//Intern Errors
IF bErrorIntern AND iErrorCode = 1 THEN
	eMessageKNXMaster := E_Message_KNXMaster.eTooMuchKNXMasters;
END_IF
//KNX Errors
IF bErrorKNX AND iErrorCode = 1 THEN
	eMessageKNXMaster := E_Message_KNXMaster.eWrong_KNX_Phys_Addr;
ELSIF bErrorKNX AND iErrorCode = 2 THEN
	eMessageKNXMaster := E_Message_KNXMaster.eWrong_KNX_Group_Addr;
ELSIF bErrorKNX AND iErrorCode = 3 THEN
	eMessageKNXMaster := E_Message_KNXMaster.eWrong_KNX_Group_Len;
ELSIF bErrorKNX AND iErrorCode = 4 THEN
	eMessageKNXMaster := E_Message_KNXMaster.eWrong_KNX_No_Filter;
ELSIF bErrorKNX AND iErrorCode = 10 THEN
	eMessageKNXMaster := E_Message_KNXMaster.eWrong_KNX_Firmware;
ELSIF bErrorKNX AND iErrorCode = 11 THEN
	eMessageKNXMaster := E_Message_KNXMaster.eWrong_KNX_Mode;
ELSIF bErrorKNX AND iErrorCode = 12 THEN
	eMessageKNXMaster := E_Message_KNXMaster.eWrong_Mode;
ELSIF bErrorKNX AND iErrorCode = 14 THEN
	eMessageKNXMaster := E_Message_KNXMaster.eWrong_KNX_Firmware_B1_Necessary;
ELSIF bErrorKNX AND iErrorCode = 15 THEN
	eMessageKNXMaster := E_Message_KNXMaster.eWrong_KNX_Firmware_B3_Necessary;
ELSIF bErrorKNX AND iErrorCode = 20 THEN
	eMessageKNXMaster := E_Message_KNXMaster.eWrong_KNX_Data_Len;
ELSIF bErrorKNX AND iErrorCode = 21 THEN
	eMessageKNXMaster := E_Message_KNXMaster.eError_KNX_Service_Not_Support;
ELSIF bErrorKNX AND iErrorCode = 30 THEN
	eMessageKNXMaster := E_Message_KNXMaster.eKL6301_TP_Toggle_Error;
ELSIF bErrorKNX AND iErrorCode = 31 THEN
	eMessageKNXMaster := E_Message_KNXMaster.eTime_Out;
ELSIF bErrorKNX AND iErrorCode = 32 THEN
	eMessageKNXMaster := E_Message_KNXMaster.eKL6301_No_Response_from_Terminal;
ELSIF bErrorKNX AND iErrorCode = 40 THEN
	eMessageKNXMaster := E_Message_KNXMaster.eError_Send_8Bit_Wrong_Scaling_Mode;
ELSIF bErrorKNX AND iErrorCode = 100 THEN
	eMessageKNXMaster := E_Message_KNXMaster.eError_KNX_Phy_Addr_Not_Support;
ELSIF bErrorKNX AND iErrorCode = 101 THEN
	eMessageKNXMaster := E_Message_KNXMaster.eError_KNX_Write_Data;
ELSIF bErrorKNX AND iErrorCode = 102 THEN
	eMessageKNXMaster := E_Message_KNXMaster.eMonitor_Mode_Len_Is_Not_Ok_Must_0;
ELSIF bErrorKNX AND iErrorCode = 103 THEN
	eMessageKNXMaster := E_Message_KNXMaster.eMonitor_Mode_Addr_Is_Not_Ok_Must_0;
ELSIF bErrorKNX AND iErrorCode = 104 THEN
	eMessageKNXMaster := E_Message_KNXMaster.eWatchdog_Error_No_Send;
ELSIF bErrorKNX AND iErrorCode = 16#0BBB THEN
	eMessageKNXMaster := E_Message_KNXMaster.eError_KNX_No_Ack;
ELSIF bErrorKNX AND iErrorCode = 16#FAFB THEN
	eMessageKNXMaster := E_Message_KNXMaster.eError_KNX_No_Com_To_TP;
ELSIF bErrorKNX AND iErrorCode = 16#0FCC THEN
	eMessageKNXMaster := E_Message_KNXMaster.eError_TP_Temp_Warning;
ELSIF bErrorKNX AND iErrorCode = 16#17CC THEN
	eMessageKNXMaster := E_Message_KNXMaster.eError_TP_Protocol_Error;
ELSIF bErrorKNX AND iErrorCode = 16#27CC THEN
	eMessageKNXMaster := E_Message_KNXMaster.eError_TP_Transmitter_Error;
ELSIF bErrorKNX AND iErrorCode = 16#47CC THEN
	eMessageKNXMaster := E_Message_KNXMaster.eError_TP_Receive_Error;
ELSIF bErrorKNX AND iErrorCode = 16#87CC THEN
	eMessageKNXMaster := E_Message_KNXMaster.eError_TP_Slave_Collision;
END_IF 

IF bWarning THEN 
	byErrorWarning := 1;
END_IF	
	IF bErrorKNX OR bErrorIntern THEN
		byErrorWarning := 2;
	END_IF

//All ok
IF NOT bErrorKNX AND NOT bErrorIntern AND NOT bWarning THEN
	eMessageKNXMaster := E_Message_KNXMaster.eAllOk;
		byErrorWarning := 0;
END_IF

END_FUNCTION_BLOCK

// ---- Bussystems/FBs Internal/MBus Master/FB_MBusMaster_Messages.TcPOU
{attribute 'conditionalshow'}
FUNCTION_BLOCK FB_MBusMaster_Messages
VAR_INPUT
	{attribute 'hide'}
	bErrorMBus							: BOOL;						//Error from the Mbus Function
	{attribute 'hide'}
	bErrorIntern						: BOOL;						//Internal Error
	{attribute 'hide'}
	bWarning							: BOOL;						//Warning from the RTU Function
	{attribute 'hide'}
	iWarningCode						: INT;						//Warning Code
	{attribute 'hide'}
	iErrorCode							: INT;						//Error Code		
END_VAR
VAR_OUTPUT
	{attribute 'hide'}
	byErrorWarning						: BYTE;						//Error Warning State
	eMessageMBusMaster					: E_Message_MBusMaster;		//Message from the MBus Master Function
END_VAR
VAR
END_VAR

//Creator : Kai Ebensperger
//Company : Lynus AG
//Date : 23.08.2021
//Version : 1.0.0.0

//With this Funciton is possible to handel the Error and Warning Codes from the MBus Master.

//Warnings
IF bWarning AND iWarningCode = 0 THEN
	eMessageMBusMaster := E_Message_MBusMaster.eNoConnectionToBackend;
END_IF

//Intern Errors
IF bErrorIntern AND iErrorCode = 1 THEN
	eMessageMBusMaster := E_Message_MBusMaster.eTooMuchMBusMasters;
END_IF
//MBus Errors
IF bErrorMBus AND iErrorCode = 101 THEN
	eMessageMBusMaster := E_Message_MBusMaster.eMBUSERROR_CIField_wrong_72hex_expected;
ELSIF bErrorMBus AND iErrorCode = 102 THEN
	eMessageMBusMaster := E_Message_MBusMaster.eMBUSERROR_no_data_received;
ELSIF bErrorMBus AND iErrorCode = 103 THEN
	eMessageMBusMaster := E_Message_MBusMaster.eMBUSERROR_error_checksum;
ELSIF bErrorMBus AND iErrorCode = 104 THEN
	eMessageMBusMaster := E_Message_MBusMaster.eMBUSERROR_error_in_head_data;
ELSIF bErrorMBus AND iErrorCode = 105 THEN
	eMessageMBusMaster := E_Message_MBusMaster.eMBUSERROR_usiAddress_over_250;
ELSIF bErrorMBus AND iErrorCode = 106 THEN
	eMessageMBusMaster := E_Message_MBusMaster.eMBUSERROR_send_error;
ELSIF bErrorMBus AND iErrorCode = 108 THEN
	eMessageMBusMaster := E_Message_MBusMaster.eMBUSERROR_received_address_wrong;
ELSIF bErrorMBus AND iErrorCode = 109 THEN
	eMessageMBusMaster := E_Message_MBusMaster.eMBUSERROR_cMBUS_MaxCom_below_1;
ELSIF bErrorMBus AND iErrorCode = 110 THEN
	eMessageMBusMaster := E_Message_MBusMaster.eMBUSERROR_iComId_over_cMBUS_MaxCom;	
ELSIF bErrorMBus AND iErrorCode = 111 THEN
	eMessageMBusMaster := E_Message_MBusMaster.eMBUSERROR_manufacturer_sign_wrong;
ELSIF bErrorMBus AND iErrorCode = 112 THEN
	eMessageMBusMaster := E_Message_MBusMaster.eMBUSERROR_baudrate_wrong;
ELSIF bErrorMBus AND iErrorCode = 113 THEN
	eMessageMBusMaster := E_Message_MBusMaster.eMBUSERROR_ReceiveBufferFull;
ELSIF bErrorMBus AND iErrorCode = 114 THEN
	eMessageMBusMaster := E_Message_MBusMaster.eMBUSERROR_E5hex_no_received;
ELSIF bErrorMBus AND iErrorCode = 115 THEN
	eMessageMBusMaster := E_Message_MBusMaster.eMBUSERROR_no_stop_character;
ELSIF bErrorMBus AND iErrorCode = 116 THEN
	eMessageMBusMaster := E_Message_MBusMaster.eMBUSERROR_length_wrong;
ELSIF bErrorMBus AND iErrorCode = 117 THEN
	eMessageMBusMaster := E_Message_MBusMaster.eMBUSERROR_wrong_terminal;
ELSIF bErrorMBus AND iErrorCode = 118 THEN
	eMessageMBusMaster := E_Message_MBusMaster.eMBUSERROR_Terminal_is_not_initialized;
ELSIF bErrorMBus AND iErrorCode = 119 THEN
	eMessageMBusMaster := E_Message_MBusMaster.eMBUSERROR_stSecAdr_udiIdNumber_wrong;
ELSIF bErrorMBus AND iErrorCode = 120 THEN
	eMessageMBusMaster := E_Message_MBusMaster.eMBUSERROR_missing_parts_telegram;
ELSIF bErrorMBus AND iErrorCode = 121 THEN
	eMessageMBusMaster := E_Message_MBusMaster.eMBUSERROR_no_stop_character_received;
ELSIF bErrorMBus AND iErrorCode = 122 THEN
	eMessageMBusMaster := E_Message_MBusMaster.eMBUSERROR_too_many_characters;
ELSIF bErrorMBus AND iErrorCode = 123 THEN
	eMessageMBusMaster := E_Message_MBusMaster.eMBUSERROR_TimeOut_FB_KL6781;
ELSIF bErrorMBus AND iErrorCode = 124 THEN
	eMessageMBusMaster := E_Message_MBusMaster.eMBUSERROR_TimeOut_MeterFB;
ELSIF bErrorMBus AND iErrorCode = 201 THEN
	eMessageMBusMaster := E_Message_MBusMaster.eMBUSERROR_COM_PARAMETERCHANGED;
ELSIF bErrorMBus AND iErrorCode = 202 THEN
	eMessageMBusMaster := E_Message_MBusMaster.eMBUSERROR_COM_TXBUFFOVERRUN;
ELSIF bErrorMBus AND iErrorCode = 210 THEN
	eMessageMBusMaster := E_Message_MBusMaster.eMBUSERROR_COM_STRINGOVERRUN;
ELSIF bErrorMBus AND iErrorCode = 211 THEN
	eMessageMBusMaster := E_Message_MBusMaster.eMBUSERROR_COM_ZEROCHARINVALID;
ELSIF bErrorMBus AND iErrorCode = 220 THEN
	eMessageMBusMaster := E_Message_MBusMaster.eMBUSERROR_COM_INVALIDPOINTER;
ELSIF bErrorMBus AND iErrorCode = 221 THEN
	eMessageMBusMaster := E_Message_MBusMaster.eMBUSERROR_COM_INVALIDRXPOINTER;
ELSIF bErrorMBus AND iErrorCode = 222 THEN
	eMessageMBusMaster := E_Message_MBusMaster.eMBUSERROR_COM_INVALIDRXLENGTH;
ELSIF bErrorMBus AND iErrorCode = 223 THEN
	eMessageMBusMaster := E_Message_MBusMaster.eMBUSERROR_COM_DATASIZEOVERRUN;
ELSIF bErrorMBus AND iErrorCode = 16#1001 THEN
	eMessageMBusMaster := E_Message_MBusMaster.eMBUSERROR_COM_INVALIDBAUDRATE;
ELSIF bErrorMBus AND iErrorCode = 16#1002 THEN
	eMessageMBusMaster := E_Message_MBusMaster.eMBUSERROR_COM_INVALIDNUMDATABITS;
ELSIF bErrorMBus AND iErrorCode = 16#1003 THEN
	eMessageMBusMaster := E_Message_MBusMaster.eMBUSERROR_COM_INVALIDNUMSTOPBITS;
ELSIF bErrorMBus AND iErrorCode = 16#1004 THEN
	eMessageMBusMaster := E_Message_MBusMaster.eMBUSERROR_COM_INVALIDPARITY;
ELSIF bErrorMBus AND iErrorCode = 16#1005 THEN
	eMessageMBusMaster := E_Message_MBusMaster.eMBUSERROR_COM_INVALIDHANDSHAKE;
ELSIF bErrorMBus AND iErrorCode = 16#1006 THEN
	eMessageMBusMaster := E_Message_MBusMaster.eMBUSERROR_COM_INVALIDNUMREGISTERS;
ELSIF bErrorMBus AND iErrorCode = 16#1007 THEN
	eMessageMBusMaster := E_Message_MBusMaster.eMBUSERROR_COM_INVALIDREGISTER;
ELSIF bErrorMBus AND iErrorCode = 16#1008 THEN
	eMessageMBusMaster := E_Message_MBusMaster.eMBUSERROR_COM_TIMEOUT;
END_IF 

IF bWarning THEN 
	byErrorWarning := 1;
END_IF	
	IF bErrorMBus OR bErrorIntern THEN
		byErrorWarning := 2;
	END_IF

//All ok
IF NOT bErrorMBus AND NOT bErrorIntern AND NOT bWarning THEN
	eMessageMBusMaster := E_Message_MBusMaster.eAllOk;
		byErrorWarning := 0;
END_IF

END_FUNCTION_BLOCK

// ---- Bussystems/FBs Internal/RTU Master/FB_MBRTUMaster_Messages.TcPOU
{attribute 'conditionalshow'}
FUNCTION_BLOCK FB_MBRTUMaster_Messages
VAR_INPUT
	{attribute 'hide'}
	bTerminalConfigured					: BOOL;						//Shows that the terminal is configured 
	{attribute 'hide'}
	bError								: BOOL;						//Error from the RTU Function
	{attribute 'hide'}
	bWarning							: BOOL;						//Warning from the RTU Function
	{attribute 'hide'}
	iWarningCode						: INT;						//Warning Code
	{attribute 'hide'}
	iErrorCode							: INT;						//Error Code		
END_VAR
VAR_OUTPUT
	{attribute 'hide'}
	byErrorWarning						: BYTE;						//Error Warning State
	eMessageMBRTUMaster					: E_Message_MBRTUMaster;	//Message from the RTU Master Function
END_VAR
VAR
END_VAR

//Creator : Kai Ebensperger
//Company : Lynus AG
//Date : 08.07.2021
//Version : 1.0.0.0

//With this Funciton is possible to handel the Error and Warning Codes from the Modbus RTU Master.

//Warnings
IF bWarning AND iWarningCode = 0 THEN 
	eMessageMBRTUMaster := E_Message_MBRTUMaster.eNoConnectionToBackend;
END_IF

//Errors
IF bError AND iErrorCode = 1 THEN
	eMessageMBRTUMaster := E_Message_MBRTUMaster.eTooMuchMBRTUMasters;
ELSIF bError AND iErrorCode = 2 THEN
	eMessageMBRTUMaster := E_Message_MBRTUMaster.eTerminalConfigurationError;
ELSIF bError AND iErrorCode = 3 THEN
	eMessageMBRTUMaster := E_Message_MBRTUMaster.eModbusErrorIllegalFunction;
ELSIF bError AND iErrorCode = 4 THEN
	eMessageMBRTUMaster := E_Message_MBRTUMaster.eModbusErrorIllegalDataAdress;
ELSIF bError AND iErrorCode = 5 THEN
	eMessageMBRTUMaster := E_Message_MBRTUMaster.eModbusErrorIllegalDataValue;
ELSIF bError AND iErrorCode = 6 THEN
	eMessageMBRTUMaster := E_Message_MBRTUMaster.eModbusErrorSlaveDeviceFailure;
ELSIF bError AND iErrorCode = 7 THEN
	eMessageMBRTUMaster := E_Message_MBRTUMaster.eModbusErrorAcknowledge;
ELSIF bError AND iErrorCode = 8 THEN
	eMessageMBRTUMaster := E_Message_MBRTUMaster.eModbusErrorSlaveDeviceBusy;
ELSIF bError AND iErrorCode = 9 THEN
	eMessageMBRTUMaster := E_Message_MBRTUMaster.eModbusErrorNegativeAcknowledge;
ELSIF bError AND iErrorCode = 10 THEN
	eMessageMBRTUMaster := E_Message_MBRTUMaster.eModbusErrorMemoryParity;
ELSIF bError AND iErrorCode = 11 THEN
	eMessageMBRTUMaster := E_Message_MBRTUMaster.eModbusErrorGatewayPathUnavailable;
ELSIF bError AND iErrorCode = 12 THEN
	eMessageMBRTUMaster := E_Message_MBRTUMaster.eModbusErrorGatewayTargetDeviceFailedToRespond;
ELSIF bError AND iErrorCode = 13 THEN
	eMessageMBRTUMaster := E_Message_MBRTUMaster.eModbusErrorCharrecTimeout;
ELSIF bError AND iErrorCode = 14 THEN
	eMessageMBRTUMaster := E_Message_MBRTUMaster.eModbusErrorIllegalDataSize;
ELSIF bError AND iErrorCode = 15 THEN
	eMessageMBRTUMaster := E_Message_MBRTUMaster.eModbusErrorIllegalDeviceAdress;
ELSIF bError AND iErrorCode = 16 THEN
	eMessageMBRTUMaster := E_Message_MBRTUMaster.eModbusErrorIllegalDestinationAdress;
ELSIF bError AND iErrorCode = 17 THEN
	eMessageMBRTUMaster := E_Message_MBRTUMaster.eModbusErrorIllegalDestinationSize;
ELSIF bError AND iErrorCode = 18 THEN
	eMessageMBRTUMaster := E_Message_MBRTUMaster.eModbusErrorNoResponse;
ELSIF bError AND iErrorCode = 19 THEN
	eMessageMBRTUMaster := E_Message_MBRTUMaster.eModbusErrorTxBufferOverrun;
ELSIF bError AND iErrorCode = 20 THEN
	eMessageMBRTUMaster := E_Message_MBRTUMaster.eModbusErrorSendTimeout;
ELSIF bError AND iErrorCode = 21 THEN
	eMessageMBRTUMaster := E_Message_MBRTUMaster.eModbusErrorDataSizeOverrun;
ELSIF bError AND iErrorCode = 22 THEN
	eMessageMBRTUMaster := E_Message_MBRTUMaster.eModbusErrorStringOverrun;
ELSIF bError AND iErrorCode = 23 THEN
	eMessageMBRTUMaster := E_Message_MBRTUMaster.eModbusErrorInvalidPointer;
ELSIF bError AND iErrorCode = 24 THEN
	eMessageMBRTUMaster := E_Message_MBRTUMaster.eModbusErrorCRC;
ELSIF bError AND iErrorCode = 25 THEN
	eMessageMBRTUMaster := E_Message_MBRTUMaster.eModbusErrorInvalidMemoryAdress;
ELSIF bError AND iErrorCode = 26 THEN
	eMessageMBRTUMaster := E_Message_MBRTUMaster.eModbusErrorTransmitBufferTooSmal;
END_IF 

IF bWarning THEN 
	byErrorWarning := 1;
END_IF	
	IF bError THEN
		byErrorWarning := 2;
	END_IF

//All ok
IF NOT bError AND NOT bWarning THEN
	eMessageMBRTUMaster := E_Message_MBRTUMaster.eAllOk;
		byErrorWarning := 0;
END_IF

//No Configuration
IF NOT bError AND NOT bTerminalConfigured THEN
	eMessageMBRTUMaster := E_Message_MBRTUMaster.eNoTerminalConfiguration;
END_IF

END_FUNCTION_BLOCK

// ---- Communicator/FBs Internal/FB_MessageRead.TcPOU
{attribute 'hide_all_locals'}
{attribute 'conditionalshow'}
FUNCTION_BLOCK FB_MessageRead
VAR_INPUT
	{attribute 'hide'}
	sReceivedMessageDoc    			: STRING(7000);																			//Received Message File from external code
	{attribute 'hide'}
	arrVarInfos						: ARRAY[1..10,1..Constants_Communicator.udiArraySizeMarkedSymobls] OF ST_Var_Info_GV;	//Infos from each plc variable		
END_VAR
VAR_OUTPUT
	{attribute 'hide'}
	stInfoFromReceivedMessage		: ST_Message_Out;																		//Output structer from the received Message file from input
	{attribute 'hide'}
	bError							: BOOL;																					//Error flag
	{attribute 'hide'}
	bMuchMoreInformationReceived	: BOOL;																					//Much more Information received
	eErrorMessage_Out				: eErrorMessage;																		//Enum with the Error states
END_VAR
VAR
	fbJsonRead					    : FB_JsonDomParser;																		//FB Json Dom reader
 	jsonDocInit  					: SJsonValue;																			//Json value
	jsonDoc		  					: SJsonValue;																			//Json value
	jsonPropID   					: SJsonValue;																			//Json value
	jsonPropValue  					: SJsonValue;																			//Json value
	jsonPropValueOut				: SJsonValue;																			//Json value
	jsonIteratorInit				: SJsonAIterator;																		//Json AIterator
	jsonIterator 					: SJsonAIterator;																		//Json AIterator
	eJsonType						: EJsonType;																			//Json Type
	arrStringValueFloat				: ARRAY[0..Constants_Communicator.bySizeOfReceivedValueArrayInJson] OF STRING(510);		//Copy received value string in this variable to check the received lengh	
	arrErrorIntern					: ARRAY[0..Constants_Communicator.bySizeOfReceivedValueArrayInJson] OF BOOL;			//Array with Error flag	
	bDetected						: BOOL;																					//True if the symbol Name is found in the internal array
	bErrorIntern					: BOOL;																					//Error flag
	byLPCheckSymbolType				: BYTE;																					//Loop to check if the symbol exist in the plc
	uiLPClearOutValues				: UINT;																					//Loop to clear output values
	udiLPCheckSymbolType			: UDINT;																				//Loop to check symbol type
	udiLPWriteValueArrayOUT			: UDINT;																				//Loop to write array value		
	udiArraySizeReceived			: UDINT;																				//Array Size from received jso	
	udiLPErrorArrayTrue				: UDINT;																				//Loop to fill the error array initial with true
	udiLPErrorArrayCheck			: UDINT;																				//Loop to check at the end of the code its 1 error flag is remained at true	
	lrFloatValue					: LREAL;																				//Float Value LREAL
	rFloatValue						: REAL;																					//Float Value REAL
	sFindMemberValue				: STRING(2);																			//Member for the value	
	(*--------------------------------------------------Not in use-----------------------------------------------------------------------*)
	jsonXMLName						: SJsonValue;																			//Json value (-)
	jsonLink						: SJsonValue;																			//Json value (l)
	jsonBaseName					: SJsonValue;																			//Json value (bn)
	jsonBaseTime					: SJsonValue;																			//Json value (bt)
	jsonBaseUnit					: SJsonValue;																			//Json value (bu)
	jsonBaseVersion					: SJsonValue;																			//Json value (bver)
	jsonBaseValue					: SJsonValue;																			//Json value (bv)
	jsonBaseSum						: SJsonValue;																			//Json value (bs)
	jsonUnit						: SJsonValue;																			//Json value (u)
	jsonTime						: SJsonValue;																			//Json value (t)
	jsonUpateTime					: SJsonValue;																			//Json value (ut)
	jsonDataValue					: SJsonValue;																			//Json value (vd)
	jsonBoolValue					: SJsonValue;																			//Json value (vb)
	jsonSum							: SJsonValue;																			//Json value (s)										
END_VAR

//Creator : Kai Ebensperger
//Company : Lynus AG
//Date : 01.04.2020
//Version : 1.0.0.0

//With this function its possible to read a json file in SenML Format
//The function produce a error if the received symbol name not exist in the internal list from the plc
//Read json files with every standart data type with single symbols and 1 dimension arrays.

(*-------------------------------------------------------------------------JSON READ--------------------------------------------------------------------------*)
//Clear output befor start to encode the received json
stInfoFromReceivedMessage.sFullSymbolName := '';
	stInfoFromReceivedMessage.sSymbolType := '';
		FOR uiLPClearOutValues := 0 TO Constants_Communicator.bySizeOfReceivedValueArrayInJson BY 1 DO
			stInfoFromReceivedMessage.arrValue[uiLPClearOutValues] := '';
				arrStringValueFloat[uiLPClearOutValues] := '';	
		END_FOR	

//Find 1 content in array because the received mesage is in SenML Format
jsonDocInit := fbJsonRead.ParseDocument(sReceivedMessageDoc);

IF jsonDocInit <> 0 THEN
	IF fbJsonRead.IsArray(jsonDocInit) AND fbJsonRead.GetArraySize(jsonDocInit) = 1 THEN
		jsonIteratorInit := fbJsonRead.ArrayBegin(jsonDocInit);
			jsonDoc := fbJsonRead.GetArrayValue(jsonIteratorInit);
	ELSE
		jsonDoc := 0;
	END_IF
ELSE
	jsonDoc := 0;
END_IF

bDetected := FALSE;

stInfoFromReceivedMessage.byReadWriteArrayNumber := LIMIT(1,stInfoFromReceivedMessage.byReadWriteArrayNumber,10);

IF jsonDoc <> 0 THEN

	jsonPropID := fbJsonRead.FindMember(jsonDoc, 'n');
	IF (jsonPropID <> 0) AND fbJsonRead.IsString(jsonPropID) THEN
	  stInfoFromReceivedMessage.sFullSymbolName := fbJsonRead.GetString(jsonPropID);
	END_IF
		//Check for accordance 
		bDetected := FALSE;
		
		IF GVL_Communicator.byNumberOfReadWriteFunction >= 1 AND GVL_Communicator.byNumberOfReadWriteFunction <= 10 THEN
			FOR byLPCheckSymbolType := 1 TO GVL_Communicator.byNumberOfReadWriteFunction BY 1 DO   
				IF GVL_Communicator.arrCounterVariableInArray[byLPCheckSymbolType] <= Constants_Communicator.udiArraySizeMarkedSymobls THEN 
					FOR udiLPCheckSymbolType := 1 TO GVL_Communicator.arrCounterVariableInArray[byLPCheckSymbolType] BY 1 DO
						IF arrVarInfos[byLPCheckSymbolType,udiLPCheckSymbolType].sFullSymbolName = stInfoFromReceivedMessage.sFullSymbolName THEN 
							stInfoFromReceivedMessage.sSymbolType := arrVarInfos[byLPCheckSymbolType,udiLPCheckSymbolType].sSymbolType; 
								stInfoFromReceivedMessage.uiSizeArray := arrVarInfos[byLPCheckSymbolType,udiLPCheckSymbolType].uiSizeArray;
									stInfoFromReceivedMessage.byReadWriteArrayNumber := byLPCheckSymbolType;	
										bDetected := TRUE;
											EXIT; 
						END_IF 
					END_FOR	
				END_IF
			END_FOR
		END_IF

			stInfoFromReceivedMessage.byReadWriteArrayNumber := LIMIT(1,stInfoFromReceivedMessage.byReadWriteArrayNumber,10);
				bErrorIntern := FALSE;
	
				IF FIND(stInfoFromReceivedMessage.sSymbolType,'STRING(30)') <> 0 OR FIND(stInfoFromReceivedMessage.sSymbolType,'OF STRING(30)') <> 0 THEN
					sFindMemberValue := 'vs';
				ELSE
					sFindMemberValue := 'v';
				END_IF
			 	
	//Single variable
	IF FIND(stInfoFromReceivedMessage.sSymbolType,'ARRAY') = 0 AND bDetected THEN
		arrErrorIntern[0] := TRUE;
			jsonPropValue := fbJsonRead.FindMember(jsonDoc,sFindMemberValue);
		IF (jsonPropValue <> 0) THEN
			eJsonType := fbJsonRead.GetType(jsonPropValue);
				//Float
				IF (stInfoFromReceivedMessage.sSymbolType = 'REAL' AND eJsonType = 6 AND fbJsonRead.IsDouble(jsonPropValue)) OR (stInfoFromReceivedMessage.sSymbolType = 'REAL' AND eJsonType = 6 AND fbJsonRead.IsInt(jsonPropValue)) THEN
					lrFloatValue := fbJsonRead.GetDouble(jsonPropValue);
						IF lrFloatValue >= -3.402823E+38 AND lrFloatValue <= 3.402823E+38 THEN  
							rFloatValue := LREAL_TO_REAL(lrFloatValue);
								IF IsFinite(F_REAL(rFloatValue)) THEN
									arrStringValueFloat[0] := REAL_TO_STRING(rFloatValue);
										IF LEN(arrStringValueFloat[0]) <= 30 THEN
											arrErrorIntern[0] := FALSE;
												stInfoFromReceivedMessage.arrValue[0] := arrStringValueFloat[0];
										END_IF
								END_IF
						END_IF
				END_IF
					IF (stInfoFromReceivedMessage.sSymbolType = 'LREAL' AND eJsonType = 6 AND fbJsonRead.IsDouble(jsonPropValue)) OR (stInfoFromReceivedMessage.sSymbolType = 'LREAL' AND eJsonType = 6 AND fbJsonRead.IsInt64(jsonPropValue)) THEN
						lrFloatValue := fbJsonRead.GetDouble(jsonPropValue);
							IF lrFloatValue >= -1.7976931348623157E+307 AND lrFloatValue <= 1.7976931348623157E+307 AND IsFinite(F_LREAL(lrFloatValue)) THEN
								arrStringValueFloat[0] := LREAL_TO_STRING(lrFloatValue);
									IF LEN(arrStringValueFloat[0]) <= 30 THEN
										arrErrorIntern[0] := FALSE;
											stInfoFromReceivedMessage.arrValue[0] := arrStringValueFloat[0];
									END_IF
							END_IF
					END_IF
						IF (stInfoFromReceivedMessage.sSymbolType = 'BOOL' OR stInfoFromReceivedMessage.sSymbolType = 'BYTE' OR stInfoFromReceivedMessage.sSymbolType = 'WORD' OR stInfoFromReceivedMessage.sSymbolType = 'DWORD' OR 
								stInfoFromReceivedMessage.sSymbolType = 'USINT' OR stInfoFromReceivedMessage.sSymbolType = 'UINT' OR stInfoFromReceivedMessage.sSymbolType = 'UDINT' OR stInfoFromReceivedMessage.sSymbolType = 'ULINT' OR 
									stInfoFromReceivedMessage.sSymbolType = 'LWORD' OR stInfoFromReceivedMessage.sSymbolType = 'TIME' OR stInfoFromReceivedMessage.sSymbolType = 'TIME_OF_DAY' OR stInfoFromReceivedMessage.sSymbolType = 'DATE' OR 
										stInfoFromReceivedMessage.sSymbolType = 'DATE_AND_TIME') AND eJsonType = 6 AND fbJsonRead.IsUint64(jsonPropValue) THEN
											arrStringValueFloat[0] := ULINT_TO_STRING(fbJsonRead.GetUint64(jsonPropValue));
												IF LEN(arrStringValueFloat[0]) <= 30 THEN arrErrorIntern[0] := FALSE; stInfoFromReceivedMessage.arrValue[0] := arrStringValueFloat[0]; END_IF
													IF (LEN(stInfoFromReceivedMessage.arrValue[0]) > 10 AND (stInfoFromReceivedMessage.sSymbolType = 'DATE_AND_TIME' OR stInfoFromReceivedMessage.sSymbolType = 'DATE')) THEN
														stInfoFromReceivedMessage.arrValue[0] := REPLACE(stInfoFromReceivedMessage.arrValue[0],'000',3,11);
													END_IF		   
							END_IF
								IF (stInfoFromReceivedMessage.sSymbolType = 'SINT' OR stInfoFromReceivedMessage.sSymbolType = 'INT' OR stInfoFromReceivedMessage.sSymbolType = 'DINT' OR stInfoFromReceivedMessage.sSymbolType = 'LINT') AND eJsonType = 6 AND fbJsonRead.IsInt64(jsonPropValue) THEN
									arrStringValueFloat[0] := LINT_TO_STRING(fbJsonRead.GetInt64(jsonPropValue));
										IF LEN(arrStringValueFloat[0]) <= 30 THEN arrErrorIntern[0] := FALSE; stInfoFromReceivedMessage.arrValue[0] := arrStringValueFloat[0]; END_IF
								END_IF
									IF stInfoFromReceivedMessage.sSymbolType = 'STRING(30)' AND eJsonType = 5 AND fbJsonRead.IsString(jsonPropValue) THEN 		
										arrStringValueFloat[0] := fbJsonRead.GetString(jsonPropValue);
											IF LEN(arrStringValueFloat[0]) <= 30 THEN arrErrorIntern[0] := FALSE; stInfoFromReceivedMessage.arrValue[0] := arrStringValueFloat[0]; END_IF
											IF LEN(arrStringValueFloat[0]) = 0 THEN arrErrorIntern[0] := FALSE; stInfoFromReceivedMessage.arrValue[0] := '#EMPTY#'; END_IF 
									END_IF
										jsonXMLName := fbJsonRead.FindMember(jsonDoc,'-');
										jsonLink := fbJsonRead.FindMember(jsonDoc,'l');
										jsonBaseName := fbJsonRead.FindMember(jsonDoc,'bn');
										jsonBaseTime := fbJsonRead.FindMember(jsonDoc,'bt');
										jsonBaseUnit := fbJsonRead.FindMember(jsonDoc,'bu');
										jsonBaseVersion := fbJsonRead.FindMember(jsonDoc,'bver');
										jsonBaseValue := fbJsonRead.FindMember(jsonDoc,'bv'); 
										jsonBaseSum := fbJsonRead.FindMember(jsonDoc,'bs'); 
										jsonUnit := fbJsonRead.FindMember(jsonDoc,'u');
										jsonTime := fbJsonRead.FindMember(jsonDoc,'t');
										jsonUpateTime := fbJsonRead.FindMember(jsonDoc,'ut');
										jsonDataValue := fbJsonRead.FindMember(jsonDoc,'vd'); 
										jsonBoolValue := fbJsonRead.FindMember(jsonDoc,'vb');  
										jsonSum := fbJsonRead.FindMember(jsonDoc,'s');  
											IF jsonXMLName <> 0 OR jsonLink <> 0 OR jsonBaseName <> 0 OR jsonBaseTime <> 0 OR jsonBaseUnit <> 0 OR jsonBaseVersion <> 0 OR jsonBaseValue <> 0 OR
												 jsonBaseSum <> 0 OR jsonUnit <> 0 OR jsonTime <> 0 OR jsonUpateTime <> 0 OR jsonDataValue <> 0 OR jsonBoolValue <> 0 OR jsonSum <> 0 THEN 
													bMuchMoreInformationReceived := TRUE; 
											ELSE 
													bMuchMoreInformationReceived := FALSE; 
											END_IF	
		END_IF
		
	ELSE
	
		IF bDetected THEN
			FOR udiLPErrorArrayTrue := 0 TO Constants_Communicator.bySizeOfReceivedValueArrayInJson BY 1 DO  
				arrErrorIntern[udiLPErrorArrayTrue] := TRUE;
			END_FOR
			//Array
			jsonPropValue := fbJsonRead.FindMember(jsonDoc,sFindMemberValue);
				IF fbJsonRead.IsArray(jsonPropValue) AND jsonPropValue <> 0 THEN
					udiArraySizeReceived := fbJsonRead.GetArraySize(jsonPropValue) - 1;
						IF udiArraySizeReceived <= Constants_Communicator.bySizeOfReceivedValueArrayInJson AND (udiArraySizeReceived + 1) = stInfoFromReceivedMessage.uiSizeArray THEN
							jsonIterator := fbJsonRead.ArrayBegin(jsonPropValue);
								FOR udiLPWriteValueArrayOUT := 0 TO udiArraySizeReceived BY 1 DO
									jsonPropValueOut := fbJsonRead.GetArrayValueByIdx(jsonPropValue,udiLPWriteValueArrayOUT);
										IF jsonPropValueOut <> 0 THEN
											eJsonType := fbJsonRead.GetType(jsonPropValueOut);
											//Float values
											IF (FIND(stInfoFromReceivedMessage.sSymbolType,'OF REAL') <> 0 AND eJsonType = 6 AND fbJsonRead.IsDouble(jsonPropValueOut)) OR (FIND(stInfoFromReceivedMessage.sSymbolType,'OF REAL') <> 0 AND eJsonType = 6 AND fbJsonRead.IsInt(jsonPropValueOut)) THEN
												lrFloatValue := fbJsonRead.GetDouble(jsonPropValueOut);
													IF lrFloatValue >= -3.402823E+38 AND lrFloatValue <= 3.402823E+38 THEN
														rFloatValue := LREAL_TO_REAL(lrFloatValue);
															IF IsFinite(F_REAL(rFloatValue)) THEN
																arrStringValueFloat[udiLPWriteValueArrayOUT] := REAL_TO_STRING(rFloatValue); 	
																	IF LEN(arrStringValueFloat[udiLPWriteValueArrayOUT]) <= 30 THEN
																		arrErrorIntern[udiLPWriteValueArrayOUT] := FALSE;
																			stInfoFromReceivedMessage.arrValue[udiLPWriteValueArrayOUT] := arrStringValueFloat[udiLPWriteValueArrayOUT];
																	END_IF
															END_IF
													END_IF
											END_IF
												//Float values
												IF (FIND(stInfoFromReceivedMessage.sSymbolType,'OF LREAL') <> 0 AND eJsonType = 6 AND fbJsonRead.IsDouble(jsonPropValueOut)) OR (FIND(stInfoFromReceivedMessage.sSymbolType,'OF LREAL') <> 0 AND eJsonType = 6 AND fbJsonRead.IsInt64(jsonPropValueOut)) THEN
													lrFloatValue := fbJsonRead.GetDouble(jsonPropValueOut);
														IF lrFloatValue >= -1.7976931348623157E+307 AND lrFloatValue <= 1.7976931348623157E+307 AND IsFinite(F_LREAL(lrFloatValue)) THEN
															arrStringValueFloat[udiLPWriteValueArrayOUT] := LREAL_TO_STRING(lrFloatValue); 	
																IF LEN(arrStringValueFloat[udiLPWriteValueArrayOUT]) <= 30 THEN
																	arrErrorIntern[udiLPWriteValueArrayOUT] := FALSE;
																		stInfoFromReceivedMessage.arrValue[udiLPWriteValueArrayOUT] := arrStringValueFloat[udiLPWriteValueArrayOUT];
																END_IF
														END_IF
												END_IF
													//only positiv values
													IF (FIND(stInfoFromReceivedMessage.sSymbolType,'OF BOOL') <> 0 OR FIND(stInfoFromReceivedMessage.sSymbolType,'OF BYTE') <> 0 OR FIND(stInfoFromReceivedMessage.sSymbolType,'OF WORD') <> 0 OR
															FIND(stInfoFromReceivedMessage.sSymbolType,'OF DWORD') <> 0 OR FIND(stInfoFromReceivedMessage.sSymbolType,'OF USINT') <> 0 OR FIND(stInfoFromReceivedMessage.sSymbolType,'OF UINT') <> 0 OR 
																FIND(stInfoFromReceivedMessage.sSymbolType,'OF UDINT') <> 0 OR FIND(stInfoFromReceivedMessage.sSymbolType,'OF ULINT') <> 0 OR FIND(stInfoFromReceivedMessage.sSymbolType,'OF LWORD') <> 0 OR
																	FIND(stInfoFromReceivedMessage.sSymbolType,'OF TIME') <> 0 OR FIND(stInfoFromReceivedMessage.sSymbolType,'OF TIME_OF_DAY') <> 0 OR FIND(stInfoFromReceivedMessage.sSymbolType,'OF DATE') <> 0 OR 
																		FIND(stInfoFromReceivedMessage.sSymbolType,'OF DATE_AND_TIME') <> 0) AND eJsonType = 6 AND fbJsonRead.IsUint64(jsonPropValueOut) THEN 
																			arrStringValueFloat[udiLPWriteValueArrayOUT] := ULINT_TO_STRING(fbJsonRead.GetUint64(jsonPropValueOut));
																				IF LEN(arrStringValueFloat[udiLPWriteValueArrayOUT]) <= 30 THEN arrErrorIntern[udiLPWriteValueArrayOUT] := FALSE; stInfoFromReceivedMessage.arrValue[udiLPWriteValueArrayOUT] := arrStringValueFloat[udiLPWriteValueArrayOUT]; END_IF
																					IF (LEN(stInfoFromReceivedMessage.arrValue[udiLPWriteValueArrayOUT]) > 10 AND (FIND(stInfoFromReceivedMessage.sSymbolType,'OF DATE_AND_TIME') <> 0 OR FIND(stInfoFromReceivedMessage.sSymbolType,'OF DATE') <> 0)) THEN
																						stInfoFromReceivedMessage.arrValue[udiLPWriteValueArrayOUT] := REPLACE(stInfoFromReceivedMessage.arrValue[udiLPWriteValueArrayOUT],'000',3,11);
																					END_IF
													END_IF
														//positiv and negativ values
														IF (FIND(stInfoFromReceivedMessage.sSymbolType,'OF SINT') <> 0 OR FIND(stInfoFromReceivedMessage.sSymbolType,'OF INT') <> 0 OR FIND(stInfoFromReceivedMessage.sSymbolType,'OF DINT') <> 0 OR
																FIND(stInfoFromReceivedMessage.sSymbolType,'OF LINT') <> 0) AND eJsonType = 6 AND fbJsonRead.IsInt64(jsonPropValueOut) THEN 
																	arrStringValueFloat[udiLPWriteValueArrayOUT] := LINT_TO_STRING(fbJsonRead.GetInt64(jsonPropValueOut));
																IF LEN(arrStringValueFloat[udiLPWriteValueArrayOUT]) <= 30 THEN arrErrorIntern[udiLPWriteValueArrayOUT] := FALSE; stInfoFromReceivedMessage.arrValue[udiLPWriteValueArrayOUT] := arrStringValueFloat[udiLPWriteValueArrayOUT]; END_IF
														END_IF
															//All string values
															IF (FIND(stInfoFromReceivedMessage.sSymbolType,'OF STRING(30)') <> 0) AND eJsonType = 5 AND fbJsonRead.IsString(jsonPropValueOut) THEN
																arrStringValueFloat[udiLPWriteValueArrayOUT] := fbJsonRead.GetString(jsonPropValueOut);
																	IF LEN(arrStringValueFloat[udiLPWriteValueArrayOUT]) <= 30 THEN arrErrorIntern[udiLPWriteValueArrayOUT] := FALSE; stInfoFromReceivedMessage.arrValue[udiLPWriteValueArrayOUT] := arrStringValueFloat[udiLPWriteValueArrayOUT]; END_IF
																	IF LEN(arrStringValueFloat[udiLPWriteValueArrayOUT]) = 0 THEN arrErrorIntern[udiLPWriteValueArrayOUT] := FALSE; stInfoFromReceivedMessage.arrValue[udiLPWriteValueArrayOUT] := '#EMPTY#'; END_IF
															END_IF
																jsonXMLName := fbJsonRead.FindMember(jsonDoc,'-');
																jsonLink := fbJsonRead.FindMember(jsonDoc,'l');
																jsonBaseName := fbJsonRead.FindMember(jsonDoc,'bn');
																jsonBaseTime := fbJsonRead.FindMember(jsonDoc,'bt');
																jsonBaseUnit := fbJsonRead.FindMember(jsonDoc,'bu');
																jsonBaseVersion := fbJsonRead.FindMember(jsonDoc,'bver');
																jsonBaseValue := fbJsonRead.FindMember(jsonDoc,'bv'); 
																jsonBaseSum := fbJsonRead.FindMember(jsonDoc,'bs'); 
																jsonUnit := fbJsonRead.FindMember(jsonDoc,'u');
																jsonTime := fbJsonRead.FindMember(jsonDoc,'t');
																jsonUpateTime := fbJsonRead.FindMember(jsonDoc,'ut');
																jsonDataValue := fbJsonRead.FindMember(jsonDoc,'vd'); 
																jsonBoolValue := fbJsonRead.FindMember(jsonDoc,'vb');  
																jsonSum := fbJsonRead.FindMember(jsonDoc,'s');  
																	IF jsonXMLName <> 0 OR jsonLink <> 0 OR jsonBaseName <> 0 OR jsonBaseTime <> 0 OR jsonBaseUnit <> 0 OR jsonBaseVersion <> 0 OR jsonBaseValue <> 0 OR
																			jsonBaseSum <> 0 OR jsonUnit <> 0 OR jsonTime <> 0 OR jsonUpateTime <> 0 OR jsonDataValue <> 0 OR jsonBoolValue <> 0 OR jsonSum <> 0 THEN 
																			bMuchMoreInformationReceived := TRUE; 
																	ELSE 
																			bMuchMoreInformationReceived := FALSE; 
																	END_IF
										END_IF							jsonIterator := fbJsonRead.NextArray(jsonIterator);		
								END_FOR	
						END_IF				
				END_IF	
		END_IF		 	
	END_IF	
END_IF

//Error flag
FOR udiLPErrorArrayCheck := 0 TO Constants_Communicator.bySizeOfReceivedValueArrayInJson BY 1 DO
	IF arrErrorIntern[udiLPErrorArrayCheck] THEN bErrorIntern := TRUE; END_IF 
END_FOR 

IF NOT bDetected OR bErrorIntern OR (jsonDoc = 0 AND sReceivedMessageDoc <> '') THEN bError := TRUE; END_IF
IF (bDetected AND NOT bErrorIntern) OR (jsonDoc = 0 AND sReceivedMessageDoc = '') THEN bError := FALSE; END_IF 

IF bErrorIntern OR bError THEN eErrorMessage_Out := eErrorMessage.eReceivedMessageWithError; 
ELSIF NOT bDetected AND bError THEN eErrorMessage_Out := eErrorMessage.eReceivedMessageIncompatibility;  
ELSE eErrorMessage_Out := eErrorMessage.eNoError; END_IF

END_FUNCTION_BLOCK

// ---- Communicator/FBs Internal/FB_MessageWrite.TcPOU
{attribute 'hide_all_locals'}
{attribute 'conditionalshow'}
FUNCTION_BLOCK FB_MessageWrite
VAR_INPUT
	{attribute 'hide'}
	bEnable							: BOOL;																			//Enable this function														
	{attribute 'hide'}
	stInfoToConvertInMessage		: ARRAY[1..10] OF ST_Message_In;												//Received raw structer to convert in message file	
END_VAR
VAR_OUTPUT
	{attribute 'hide'}
	sMessageDocToWrite  	 		: STRING(7000);																	//Message file from raw input structer
	{attribute 'hide'}
	bError							: BOOL;																			//Error Message write
	{attribute 'hide'}
	bDone							: BOOL;
	eErrorMessage_Out				: eErrorMessage;																//Error Message
END_VAR
VAR
	fbJsonWrite     				: FB_JsonSaxWriter;																//FB Sax Writer
	arrFind							: ARRAY[1..2] OF INT;															//Help variable for string functions
	byLPPrepearJson					: BYTE;																			//Loop to prepear the json with input settings
	iStatePrepearJson				: INT;																			//State Maschine
	uiSizeArray						: UINT;																			//Array Size
	uiValueLower					: UINT;																			//Lower value from array size
	uiValueHigher					: UINT;																			//Higher value from array size
	uiLPWriteValueArrayIN			: UINT;																			//Loop to write array value		
	sJsonDocToWriteInt   			: STRING(255);																	//Json file from raw input structer	
	sAddKeyValue					: STRING(2);																	//Key for the Value in the string	
	rNumer							: REAL;																			//Real number to check for valid value
	lrNumer							: LREAL;																		//LReal number to check for valid value
END_VAR

//Creator : Kai Ebensperger
//Company : Lynus AG
//Date : 01.04.2020
//Version : 1.0.0.0

//With this function its possible to create a json file in SenML Format
//Create json files with every standart data type with single symbols and 1 dimension arrays.

CASE iStatePrepearJson OF

	0://Start if somthing is inside the Array
	bDone := FALSE;
	
	IF GVL_Communicator.byNumberOfReadWriteFunction >= 1 AND GVL_Communicator.byNumberOfReadWriteFunction <= 10 AND bEnable THEN
		FOR byLPPrepearJson := 1 TO GVL_Communicator.byNumberOfReadWriteFunction BY 1 DO
			IF FIND(stInfoToConvertInMessage[byLPPrepearJson].sSymbolType,'BOOL') = 1 OR FIND(stInfoToConvertInMessage[byLPPrepearJson].sSymbolType,'BYTE') = 1 OR FIND(stInfoToConvertInMessage[byLPPrepearJson].sSymbolType,'WORD') = 1 OR FIND(stInfoToConvertInMessage[byLPPrepearJson].sSymbolType,'DWORD') = 1 OR
				FIND(stInfoToConvertInMessage[byLPPrepearJson].sSymbolType,'SINT') = 1 OR FIND(stInfoToConvertInMessage[byLPPrepearJson].sSymbolType,'USINT') = 1 OR FIND(stInfoToConvertInMessage[byLPPrepearJson].sSymbolType,'INT') = 1 OR FIND(stInfoToConvertInMessage[byLPPrepearJson].sSymbolType,'UINT') = 1 OR
					FIND(stInfoToConvertInMessage[byLPPrepearJson].sSymbolType,'DINT') = 1 OR FIND(stInfoToConvertInMessage[byLPPrepearJson].sSymbolType,'UDINT') = 1 OR FIND(stInfoToConvertInMessage[byLPPrepearJson].sSymbolType,'LINT') = 1 OR FIND(stInfoToConvertInMessage[byLPPrepearJson].sSymbolType,'ULINT') = 1 OR 
						FIND(stInfoToConvertInMessage[byLPPrepearJson].sSymbolType,'REAL') = 1 OR FIND(stInfoToConvertInMessage[byLPPrepearJson].sSymbolType,'LREAL') = 1 OR FIND(stInfoToConvertInMessage[byLPPrepearJson].sSymbolType,'STRING(30)') = 1 OR FIND(stInfoToConvertInMessage[byLPPrepearJson].sSymbolType,'TIME') = 1 OR
							FIND(stInfoToConvertInMessage[byLPPrepearJson].sSymbolType,'TIME_OF_DAY') = 1 OR FIND(stInfoToConvertInMessage[byLPPrepearJson].sSymbolType,'DATE') = 1 OR FIND(stInfoToConvertInMessage[byLPPrepearJson].sSymbolType,'DATE_AND_TIME') = 1 OR FIND(stInfoToConvertInMessage[byLPPrepearJson].sSymbolType,'LWORD') = 1 OR 
								FIND(stInfoToConvertInMessage[byLPPrepearJson].sSymbolType,'ARRAY') = 1 THEN
				bError := FALSE;
				eErrorMessage_Out := eErrorMessage.eNoError;
				fbJsonWrite.StartArray();	
				iStatePrepearJson := 1;	
				EXIT;	
			END_IF
		END_FOR
	END_IF
		
	1://Prepear Json
		IF GVL_Communicator.byNumberOfReadWriteFunction >= 1 AND GVL_Communicator.byNumberOfReadWriteFunction <= 10 THEN
			FOR byLPPrepearJson := 1 TO GVL_Communicator.byNumberOfReadWriteFunction BY 1 DO
				//Change key for the value
				IF FIND(stInfoToConvertInMessage[byLPPrepearJson].sSymbolType,'STRING(30)') <> 0 OR FIND(stInfoToConvertInMessage[byLPPrepearJson].sSymbolType,'OF STRING(30)') <> 0 THEN
					sAddKeyValue := 'vs';
				ELSE
					sAddKeyValue := 'v';
				END_IF
				
				//Check it is a single standard variable
				IF FIND(stInfoToConvertInMessage[byLPPrepearJson].sSymbolType,'BOOL') = 1 OR FIND(stInfoToConvertInMessage[byLPPrepearJson].sSymbolType,'BYTE') = 1 OR FIND(stInfoToConvertInMessage[byLPPrepearJson].sSymbolType,'WORD') = 1 OR FIND(stInfoToConvertInMessage[byLPPrepearJson].sSymbolType,'DWORD') = 1 OR
					FIND(stInfoToConvertInMessage[byLPPrepearJson].sSymbolType,'SINT') = 1 OR FIND(stInfoToConvertInMessage[byLPPrepearJson].sSymbolType,'USINT') = 1 OR FIND(stInfoToConvertInMessage[byLPPrepearJson].sSymbolType,'INT') = 1 OR FIND(stInfoToConvertInMessage[byLPPrepearJson].sSymbolType,'UINT') = 1 OR
						FIND(stInfoToConvertInMessage[byLPPrepearJson].sSymbolType,'DINT') = 1 OR FIND(stInfoToConvertInMessage[byLPPrepearJson].sSymbolType,'UDINT') = 1 OR FIND(stInfoToConvertInMessage[byLPPrepearJson].sSymbolType,'LINT') = 1 OR FIND(stInfoToConvertInMessage[byLPPrepearJson].sSymbolType,'ULINT') = 1 OR 
							FIND(stInfoToConvertInMessage[byLPPrepearJson].sSymbolType,'REAL') = 1 OR FIND(stInfoToConvertInMessage[byLPPrepearJson].sSymbolType,'LREAL') = 1 OR FIND(stInfoToConvertInMessage[byLPPrepearJson].sSymbolType,'STRING(30)') = 1 OR FIND(stInfoToConvertInMessage[byLPPrepearJson].sSymbolType,'TIME') = 1 OR
								FIND(stInfoToConvertInMessage[byLPPrepearJson].sSymbolType,'TIME_OF_DAY') = 1 OR FIND(stInfoToConvertInMessage[byLPPrepearJson].sSymbolType,'DATE') = 1 OR FIND(stInfoToConvertInMessage[byLPPrepearJson].sSymbolType,'DATE_AND_TIME') = 1 OR FIND(stInfoToConvertInMessage[byLPPrepearJson].sSymbolType,'LWORD') = 1 THEN
					fbJsonWrite.StartObject();
					fbJsonWrite.AddKey('n');
					fbJsonWrite.AddString(stInfoToConvertInMessage[byLPPrepearJson].sFullSymbolName);
					fbJsonWrite.AddKey(sAddKeyValue);
					IF stInfoToConvertInMessage[byLPPrepearJson].sSymbolType = 'BOOL' THEN fbJsonWrite.AddUdint(STRING_TO_BYTE(stInfoToConvertInMessage[byLPPrepearJson].arrValue[1])); END_IF 
					IF stInfoToConvertInMessage[byLPPrepearJson].sSymbolType = 'BYTE' THEN fbJsonWrite.AddUdint(STRING_TO_BYTE(stInfoToConvertInMessage[byLPPrepearJson].arrValue[1])); END_IF 
					IF stInfoToConvertInMessage[byLPPrepearJson].sSymbolType = 'WORD' THEN fbJsonWrite.AddUdint(STRING_TO_WORD(stInfoToConvertInMessage[byLPPrepearJson].arrValue[1])); END_IF 
					IF stInfoToConvertInMessage[byLPPrepearJson].sSymbolType = 'DWORD' THEN fbJsonWrite.AddUdint(STRING_TO_DWORD(stInfoToConvertInMessage[byLPPrepearJson].arrValue[1])); END_IF 
					IF stInfoToConvertInMessage[byLPPrepearJson].sSymbolType = 'SINT' THEN fbJsonWrite.AddDint(STRING_TO_SINT(stInfoToConvertInMessage[byLPPrepearJson].arrValue[1])); END_IF 
					IF stInfoToConvertInMessage[byLPPrepearJson].sSymbolType = 'USINT' THEN fbJsonWrite.AddUdint(STRING_TO_USINT(stInfoToConvertInMessage[byLPPrepearJson].arrValue[1])); END_IF 
					IF stInfoToConvertInMessage[byLPPrepearJson].sSymbolType = 'INT' THEN fbJsonWrite.AddDint(STRING_TO_INT(stInfoToConvertInMessage[byLPPrepearJson].arrValue[1])); END_IF
					IF stInfoToConvertInMessage[byLPPrepearJson].sSymbolType = 'UINT' THEN fbJsonWrite.AddUdint(STRING_TO_UINT(stInfoToConvertInMessage[byLPPrepearJson].arrValue[1])); END_IF
					IF stInfoToConvertInMessage[byLPPrepearJson].sSymbolType = 'DINT' THEN fbJsonWrite.AddDint(STRING_TO_DINT(stInfoToConvertInMessage[byLPPrepearJson].arrValue[1])); END_IF
					IF stInfoToConvertInMessage[byLPPrepearJson].sSymbolType = 'UDINT' THEN fbJsonWrite.AddUdint(STRING_TO_UDINT(stInfoToConvertInMessage[byLPPrepearJson].arrValue[1])); END_IF
					IF stInfoToConvertInMessage[byLPPrepearJson].sSymbolType = 'LINT' THEN fbJsonWrite.AddLint(STRING_TO_LINT(stInfoToConvertInMessage[byLPPrepearJson].arrValue[1])); END_IF
					IF stInfoToConvertInMessage[byLPPrepearJson].sSymbolType = 'ULINT' THEN fbJsonWrite.AddUlint(STRING_TO_ULINT(stInfoToConvertInMessage[byLPPrepearJson].arrValue[1])); END_IF
					IF stInfoToConvertInMessage[byLPPrepearJson].sSymbolType = 'REAL' THEN
						rNumer := STRING_TO_REAL(stInfoToConvertInMessage[byLPPrepearJson].arrValue[1]); 
							IF IsFinite(F_REAL(rNumer)) THEN
								fbJsonWrite.AddReal(rNumer); 
							ELSE
								bError := TRUE;
									eErrorMessage_Out := eErrorMessage.eCreatedMessageWithError;	
							END_IF
					END_IF
					IF stInfoToConvertInMessage[byLPPrepearJson].sSymbolType = 'LREAL' THEN 
						lrNumer := STRING_TO_LREAL(stInfoToConvertInMessage[byLPPrepearJson].arrValue[1]);
							IF IsFinite(F_LREAL(lrNumer)) THEN	
								fbJsonWrite.AddLreal(lrNumer); 
							ELSE
								bError := TRUE;
									eErrorMessage_Out := eErrorMessage.eCreatedMessageWithError;
							END_IF
					END_IF
					IF stInfoToConvertInMessage[byLPPrepearJson].sSymbolType = 'STRING(30)' THEN fbJsonWrite.AddString(stInfoToConvertInMessage[byLPPrepearJson].arrValue[1]); END_IF
					IF stInfoToConvertInMessage[byLPPrepearJson].sSymbolType = 'TIME' THEN fbJsonWrite.AddUdint(STRING_TO_UDINT(stInfoToConvertInMessage[byLPPrepearJson].arrValue[1])); END_IF
					IF stInfoToConvertInMessage[byLPPrepearJson].sSymbolType = 'TIME_OF_DAY' THEN fbJsonWrite.AddUdint(STRING_TO_UDINT(stInfoToConvertInMessage[byLPPrepearJson].arrValue[1])); END_IF
					IF stInfoToConvertInMessage[byLPPrepearJson].sSymbolType = 'DATE' THEN fbJsonWrite.AddUdint(STRING_TO_UDINT(stInfoToConvertInMessage[byLPPrepearJson].arrValue[1])); END_IF
					IF stInfoToConvertInMessage[byLPPrepearJson].sSymbolType = 'DATE_AND_TIME' THEN fbJsonWrite.AddUdint(STRING_TO_UDINT(stInfoToConvertInMessage[byLPPrepearJson].arrValue[1])); END_IF
					IF stInfoToConvertInMessage[byLPPrepearJson].sSymbolType = 'LWORD' THEN fbJsonWrite.AddUlint(STRING_TO_LWORD(stInfoToConvertInMessage[byLPPrepearJson].arrValue[1])); END_IF
					fbJsonWrite.AddKey('u');
					fbJsonWrite.AddString(stInfoToConvertInMessage[byLPPrepearJson].sSymbolUnit);
					fbJsonWrite.EndObject();
						rNumer := 0;
						lrNumer := 0;
				END_IF
					IF FIND(stInfoToConvertInMessage[byLPPrepearJson].sSymbolType,'ARRAY') = 1 THEN
						//Prepear json for array with standard variable	
						//detect array size
						arrFind[1] := FIND(stInfoToConvertInMessage[byLPPrepearJson].sSymbolType,'[');
						uiValueLower := STRING_TO_UINT(MID(stInfoToConvertInMessage[byLPPrepearJson].sSymbolType,1,arrFind[1] + 1));
						arrFind[2] := FIND(stInfoToConvertInMessage[byLPPrepearJson].sSymbolType,']');
							IF arrFind[1] = 7 AND arrFind[2] = 12 THEN
								uiValueHigher := STRING_TO_UINT(MID(stInfoToConvertInMessage[byLPPrepearJson].sSymbolType,1,arrFind[2] - 1));
							ELSIF arrFind[1] = 7 AND arrFind[2] = 13 THEN
								uiValueHigher := STRING_TO_UINT(MID(stInfoToConvertInMessage[byLPPrepearJson].sSymbolType,2,arrFind[2] - 2));
							ELSIF arrFind[1] = 7 AND arrFind[2] = 14 THEN
								uiValueHigher := STRING_TO_UINT(MID(stInfoToConvertInMessage[byLPPrepearJson].sSymbolType,3,arrFind[2] - 3));
							END_IF	
								uiSizeArray := (uiValueHigher - uiValueLower) + 1;
						
						fbJsonWrite.StartObject();
						fbJsonWrite.AddKey('n');
						fbJsonWrite.AddString(stInfoToConvertInMessage[byLPPrepearJson].sFullSymbolName);
						fbJsonWrite.AddKey(sAddKeyValue);
						fbJsonWrite.StartArray();
						IF uiSizeArray <= Constants_Communicator.bySizeOfValueArray THEN
							FOR uiLPWriteValueArrayIN := 1 TO uiSizeArray BY 1 DO
								IF FIND(stInfoToConvertInMessage[byLPPrepearJson].sSymbolType,'OF STRING(30)') <> 0 THEN 
									fbJsonWrite.AddString(stInfoToConvertInMessage[byLPPrepearJson].arrValue[uiLPWriteValueArrayIN]);
								ELSIF FIND(stInfoToConvertInMessage[byLPPrepearJson].sSymbolType,'OF REAL') <> 0 THEN
									rNumer := STRING_TO_REAL(stInfoToConvertInMessage[byLPPrepearJson].arrValue[uiLPWriteValueArrayIN]); 
										IF IsFinite(F_REAL(rNumer)) THEN  
											fbJsonWrite.AddReal(rNumer);
										ELSE
											bError := TRUE;
												eErrorMessage_Out := eErrorMessage.eCreatedMessageWithError;
										END_IF
								ELSIF FIND(stInfoToConvertInMessage[byLPPrepearJson].sSymbolType,'OF LREAL') <> 0 THEN
									lrNumer := STRING_TO_LREAL(stInfoToConvertInMessage[byLPPrepearJson].arrValue[uiLPWriteValueArrayIN]); 
										IF IsFinite(F_LREAL(lrNumer)) THEN  
											fbJsonWrite.AddLreal(lrNumer);
										ELSE
											bError := TRUE;
												eErrorMessage_Out := eErrorMessage.eCreatedMessageWithError;
										END_IF
								ELSE
										fbJsonWrite.AddRawArray(stInfoToConvertInMessage[byLPPrepearJson].arrValue[uiLPWriteValueArrayIN]);
								END_IF
							END_FOR
						ELSE
							bError := TRUE;
						END_IF
						fbJsonWrite.EndArray();
						fbJsonWrite.AddKey('u');
						fbJsonWrite.AddString(stInfoToConvertInMessage[byLPPrepearJson].sSymbolUnit);
						fbJsonWrite.EndObject();
							rNumer := 0;
							lrNumer := 0;
					END_IF
			END_FOR	
		END_IF
			//Json is ready		
			fbJsonWrite.EndArray();
			sJsonDocToWriteInt := fbJsonWrite.GetDocument();
			fbJsonWrite.CopyDocument(sMessageDocToWrite, SIZEOF(sMessageDocToWrite));
			fbJsonWrite.ResetDocument();
				bDone := TRUE;
				//Error when in 1 step the old messege is included befor the new one is ready
				IF LEN2(ADR(sMessageDocToWrite)) <= 2 THEN bError := TRUE; END_IF 
					iStatePrepearJson := 0;			
END_CASE

END_FUNCTION_BLOCK

// ---- Communicator/FBs Internal/FB_ParsDocument.TcPOU
{attribute 'hide_all_locals'}
{attribute 'conditionalshow'}
FUNCTION_BLOCK FB_ParsDocument
VAR_INPUT
	{attribute 'hide'}
	bRead								: BOOL;																											//Rising edge start the function
	{attribute 'hide'}
	bStop								: BOOL;																											//Stop the parsing in this Function
	{attribute 'hide'}
	eSavePositionTMCFile				: eSavePositionFile;																							//Save position from tmc file
END_VAR
VAR_OUTPUT
	{attribute 'hide'}
	arrContentOfDocument				: ARRAY[1..Constants_Communicator.uiArraySizeOfSubItems] OF ST_Content_Of_Document;								//Struct with content of the symbols
	{attribute 'hide'}
	uiFoundItems						: UINT;																											//Found Items in the Document
	{attribute 'hide'}
	bError								: BOOL;																											//Error state
	{attribute 'hide'}
	udiErrorCode						: UDINT;																										//Error Code
	{attribute 'hide'}
	bBusy								: BOOL;																											//Busy state
	{attribute 'hide'}
	bDone								: BOOL;																											//True if the function was successful
	{attribute 'hide'}
	byProgress							: BYTE;																											//Progress
	{attribute 'hide'}
	sSymbolNameWithError				: STRING(97);																									//Smbol Type with Error
END_VAR
VAR
	fbFileOpen							: FB_FileOpen;																									//Function for open the document
	fbFileGet							: FB_FileGets;																									//Function for read out the content from the open document
	fbFileTell							: FB_FileTell;																									//Function to check the actual position in the open file
	fbFileSeek							: FB_FileSeek;																									//Function to go to the end of the file
	fbFileClose							: FB_FileClose;																									//Function to close the document after complete read out
	FPStart								: R_TRIG;																										//Internal risinge edge
	FPStop								: R_TRIG;																										//Internal risinge edge
	FPErrorOpen							: R_TRIG;																										//Internal risinge edge
	FPErrorGet							: R_TRIG;																										//Internal risinge edge
	FPErrorTell							: R_TRIG;																										//Internal risinge edge
	FPErrorSeek							: R_TRIG;																										//Internal risinge edge
	FPErrorClose						: R_TRIG;																										//Internal risinge edge
	FPState2							: R_TRIG;																										//Internal risinge edge
	timTimout							: TON;																											//Timout timer for state maschine
	arrCheckListForNestedSymbols		: ARRAY[1..Constants_Communicator.uiArraySizeOfSubItems] OF STRING(48); 										//Check List for nestend symbols in an function block or a struct 												
	arrNumberForLPCheckIdentSymbols		: ARRAY[1..4] OF UINT;																							//Loop in 4 pices that code works on small plc 
	bRestOfDescriptionInNextLine		: BOOL;																											//True if in 1 received line from the GET function is not the complete description
	bNoNewDescription					: BOOL;																											//True if in 1 line is not the complete descrption and the rest from the line is '', then in the next step we have the complete description but no content. Then with that variable we save the description for next step
	bSymbolNameFound					: BOOL;																											//True if the symbol was found in the file, after that check the subitems
	bNotGet								: BOOL;																											//If the rest from the old line is concat with the new line and its done, read the rest from the new line befor start a new get  
	bFBOrStructDetected					: BOOL;																											//True if a struct or a fb is detected
	bEnumDetected						: BOOL;																											//True if a enum is detected
	bWaitForFB							: BOOL;																											//Wait than its possible that the symbol is a Function Block
	bDeleteStep3						: BOOL;																											//True if in Step 3 a pice of the received line is deleted
	byCounterWaitInStep					: BYTE;																											//Cycles that are serviced in steps
	uiSubItemArrayInProgress			: UINT;																											//Array which is in progress for save content of the subitems
	uiLPClearStruct						: UINT;																											//Loop to clear the struct at the beginning from the state maschine
	uiCounterWantedSymbolInProgress		: UINT;																											//Counted symbols with right comment
	uiCounterClearStruct				: UINT;																											//Counter to clear struct
	uiDimensionArray					: UINT;																											//Dimension of array
	uiCounterInProgressFromDocument		: UINT;																											//Counter that rear out the array from foundet symbols from the document
	uiCounterListForFBorStruct			: UINT;																											//Counter to write internal structs to check if they are available
	uiCounterCheckSubItemsInContentOfDoc: UINT;																											//Counter to ckeck if the Subitems are in the content of the document
	uiCounterFBorStruct					: UINT;																											//Counter to check for no Standart Datatyp in found symbols
	uiLPCheckIdentSymbols				: UINT;																											//Check ident internal symbols
	uiLPCkeckContentInSubItems			: UINT;																											//Loop to check the content if in a Subitem is a other subitem includet
	uiCounterCkeckContenInSubItems_1	: UINT;																											//Check if in the subitems in the structs or Functionblocks is not more than 1 extra Subitem (Number of the actual Symbol)
	uiCounterCkeckContenInSubItems_2	: UINT;																											//Check if in the subitems in the structs or Functionblocks is not more than 1 extra Subitem (Number of included Symbol Types)
	iFindBegin							: INT;																											//Find beginn position of content in the document
	iFindEnd							: INT;																											//Find end position of content in the document
	iFindBeginComment					: INT;																											//Find beginn position of the comment in the document from the subitems
	iFindEndComment						: INT;																											//Find end position of the comment in the document from the subitems	
	iLenghComment						: INT;																											//Lenght of the comment in the document from the subitems
	iStateParseDocument					: INT;																											//State of the state maschine
	diEndPositionInDocument				: DINT;																											//End of the position from the open file
	uliSizeOfString						: ULINT;																										//Size from the String in the Sub Item
	sLine								: T_MaxString;																									//Actual line with content from the document
	sLineRest							: T_MaxString;																									//Rest from the actual line if not all information from the contetn is included
	sDescription						: T_MaxString;																									//Description from the type that was found in the document
	sSymbolName							: T_MaxString;																									//Symbol Name to check that the lenght from the string is ok
	sNameSubItem						: T_MaxString;																									//Name from subitem to check that the lenght from the string is ok
	sNameSubItemOld						: T_MaxString;																									//Old name from SubItem that we can clean old information from previos SubItem
	sTypeSubItem						: T_MaxString;																									//Type from the sub item
	sTextEnum							: T_MaxString;																									//Text from the Enum
	sIndexEnum							: T_MaxString;																									//Index of the value fromt the enum
	sComment							: T_MaxString;																									//Comment from the subitem in progress
	sValue								: T_MaxString;																									//Value from symbol
	sLBound								: T_MaxString;																									//Lower Bound from array
	sElements							: T_MaxString;																									//Elements in array
	sUnit								: T_MaxString;																									//Unit from the subitme in progress
END_VAR

//Creator : Kai Ebensperger
//Company : Lynus AG
//Date : 04.05.2020
//Version : 2.0.0.0

//With this function is possible to read out the tmc file from a project to find out all information from structs,fb and enums.

FPStart(CLK:= bRead, Q=> );
	FPStop(CLK:= bStop, Q=> );

IF FPStart.Q AND iStateParseDocument = 0 THEN iStateParseDocument := - 5; END_IF
	IF FPStop.Q THEN iStateParseDocument := 100; END_IF

FPState2(CLK:= iStateParseDocument = 2, Q=> );

IF iStateParseDocument = -5 OR iStateParseDocument = 0 OR iStateParseDocument = 101 OR iStateParseDocument = 102 OR iStateParseDocument = 103 OR iStateParseDocument = 104 OR iStateParseDocument = 105 OR FPState2.Q THEN timTimout.IN := FALSE; ELSE timTimout.IN := TRUE; END_IF 
	timTimout(IN:= , PT:= T#2S, Q=> , ET=> );

CASE iStateParseDocument OF
	
	-5://Reset struct and check the size of wanted symbols
		uiCounterClearStruct := uiCounterClearStruct + 1;
			uiCounterClearStruct := LIMIT(1,uiCounterClearStruct,Constants_Communicator.uiArraySizeOfSubItems);
	
		arrContentOfDocument[uiCounterClearStruct].sSymbolName := '';
			arrContentOfDocument[uiCounterClearStruct].eSymbolType := eSymbolTypeFromDocument.eNoInformation;
				arrCheckListForNestedSymbols[uiCounterClearStruct] := '';
					FOR uiLPClearStruct := 1 TO Constants_Communicator.uiArraySizeOfMarkedSubItems BY 1 DO
						arrContentOfDocument[uiCounterClearStruct].arrSubItemName[uiLPClearStruct] := '';
							arrContentOfDocument[uiCounterClearStruct].arrSubItemSymbolType[uiLPClearStruct] := '';	
								arrContentOfDocument[uiCounterClearStruct].arrSubItemTextEnum[uiLPClearStruct] := '';
									arrContentOfDocument[uiCounterClearStruct].arrSubItemIndexEnum[uiLPClearStruct] := '';
										arrContentOfDocument[uiCounterClearStruct].arrSubItemUnit[uiLPClearStruct] := '';	
					END_FOR 	
		
		bError := FALSE;
			udiErrorCode := 0;	
				bBusy := TRUE;
					bDone := FALSE;
						sSymbolNameWithError := '';
							uiCounterWantedSymbolInProgress := 1;
								diEndPositionInDocument := 0;
									byProgress := 0;	
										uiFoundItems := 0;	
				
		IF uiCounterClearStruct >= Constants_Communicator.uiArraySizeOfSubItems THEN 
			iStateParseDocument := - 4;	
				uiCounterClearStruct := 0;
		END_IF
									
	-4://Open File to Check the Size from the file
		fbFileOpen.bExecute := TRUE;

		byCounterWaitInStep := byCounterWaitInStep + 1;
		
		IF NOT fbFileOpen.bBusy AND NOT fbFileOpen.bError AND byCounterWaitInStep >= 2 THEN iStateParseDocument := - 3; fbFileOpen.bExecute := FALSE; byCounterWaitInStep := 0; END_IF	

		IF FPErrorOpen.Q OR timTimout.Q THEN 
			iStateParseDocument := 200; 
				IF FPErrorOpen.Q THEN udiErrorCode := 105; END_IF 
					IF timTimout.Q THEN udiErrorCode := 100; END_IF 
		END_IF
						
	-3://Go to the End from the Line
		fbFileSeek.bExecute := TRUE;

		byCounterWaitInStep := byCounterWaitInStep + 1;	
		
		IF NOT fbFileSeek.bBusy AND NOT fbFileSeek.bError AND byCounterWaitInStep >= 2 THEN iStateParseDocument := - 2; fbFileSeek.bExecute := FALSE; byCounterWaitInStep := 0; END_IF	

		IF FPErrorSeek.Q OR timTimout.Q THEN 
			iStateParseDocument := 200; 
				IF FPErrorSeek.Q THEN udiErrorCode := 114; END_IF 
					IF timTimout.Q THEN udiErrorCode := 100; END_IF 
		END_IF
		
	-2://Check Position in file to calculate the progress state 0-100%
		fbFileTell.bExecute := TRUE;

		byCounterWaitInStep := byCounterWaitInStep + 1;
		
		IF NOT fbFileTell.bBusy AND NOT fbFileTell.bError AND byCounterWaitInStep >= 2 THEN iStateParseDocument := - 1; fbFileTell.bExecute := FALSE; byCounterWaitInStep := 0; diEndPositionInDocument := fbFileTell.nSeekPos; END_IF
					
		IF FPErrorTell.Q OR timTimout.Q THEN 
			iStateParseDocument := 200; 
				IF FPErrorTell.Q THEN udiErrorCode := 113; END_IF 
					IF timTimout.Q THEN udiErrorCode := 100; END_IF 
		END_IF 		
	
	-1://Close the file
		fbFileClose.bExecute := TRUE;

		byCounterWaitInStep := byCounterWaitInStep + 1; 
		
		IF NOT fbFileClose.bBusy AND NOT fbFileClose.bError AND byCounterWaitInStep >= 2 THEN iStateParseDocument := 1; fbFileClose.bExecute := FALSE; byCounterWaitInStep := 0; END_IF	
		
		IF FPErrorClose.Q OR timTimout.Q THEN 
			iStateParseDocument := 200; 
				IF FPErrorClose.Q THEN udiErrorCode := 107; END_IF 
					IF timTimout.Q THEN udiErrorCode := 100; END_IF 
		END_IF 		
		
	0://Init step and set all Variables to default value for next start
		byCounterWaitInStep := 0; iFindBegin := 0; iFindEnd := 0; uiSubItemArrayInProgress := 0; sLine := ''; sLineRest := ''; sDescription := ''; sSymbolName := ''; sNameSubItem := ''; sTextEnum := ''; sIndexEnum := ''; sComment := '';
			sTypeSubItem := ''; iLenghComment := 0; sValue := ''; uiCounterClearStruct := 0; sLBound := ''; sElements := ''; uiDimensionArray := 0; uliSizeOfString := 0; sNameSubItemOld := ''; sUnit := '';
				bRestOfDescriptionInNextLine := FALSE; bSymbolNameFound := FALSE; fbFileOpen.bExecute := FALSE; fbfileGet.bExecute := FALSE; fbFileClose.bExecute := FALSE; bFBOrStructDetected := FALSE; bWaitForFB := FALSE; bDeleteStep3 := FALSE;
					bNotGet := FALSE; bRead := FALSE; bBusy := FALSE; bNoNewDescription := FALSE; bEnumDetected := FALSE; uiCounterWantedSymbolInProgress := 0; uiCounterFBorStruct := 0;	
						uiCounterInProgressFromDocument := 0; uiCounterListForFBorStruct := 0; fbFileTell.bExecute := FALSE; fbFileSeek.bExecute := FALSE; uiCounterCheckSubItemsInContentOfDoc := 0;
							arrNumberForLPCheckIdentSymbols[1] := 0; arrNumberForLPCheckIdentSymbols[2] := 0; arrNumberForLPCheckIdentSymbols[3] := 0; arrNumberForLPCheckIdentSymbols[4] := 0; uiCounterCkeckContenInSubItems_1 := 0;
								uiCounterCkeckContenInSubItems_2 := 0;		

	1://File open
		fbFileOpen.bExecute := TRUE;

		byCounterWaitInStep := byCounterWaitInStep + 1;
		
		IF NOT fbFileOpen.bBusy AND NOT fbFileOpen.bError AND byCounterWaitInStep >= 2 THEN iStateParseDocument := 2; fbFileOpen.bExecute := FALSE; byCounterWaitInStep := 0; END_IF	

		IF FPErrorOpen.Q OR timTimout.Q THEN 
			iStateParseDocument := 200; 
				IF FPErrorOpen.Q THEN udiErrorCode := 105; END_IF 
					IF timTimout.Q THEN udiErrorCode := 100; END_IF 
		END_IF
		
	2://Get line
		IF NOT bNotGet THEN fbFileGet.bExecute := TRUE;	END_IF	
		
		byCounterWaitInStep := byCounterWaitInStep + 1;
		
		IF NOT fbFileGet.bBusy AND NOT fbFileGet.bError AND byCounterWaitInStep >= 2 AND NOT bRestOfDescriptionInNextLine AND NOT bNotGet THEN 
			iStateParseDocument := 3; fbfileGet.bExecute := FALSE; byCounterWaitInStep := 0;
				sLine := fbfileGet.sLine; 
		END_IF	
			IF NOT fbFileGet.bBusy AND NOT fbFileGet.bError AND byCounterWaitInStep >= 2 AND bRestOfDescriptionInNextLine AND NOT bNotGet THEN 
				IF (FIND(fbFileGet.sLine,'>')) + LEN(sLineRest) <= 255 THEN 
					IF FIND(fbFileGet.sLine,'>') <> 0 THEN sLine := CONCAT(sLineRest,LEFT(fbFileGet.sLine,FIND(fbFileGet.sLine,'>'))); bNotGet := TRUE; END_IF
				ELSE
					iStateParseDocument := 200; udiErrorCode := 101;
				END_IF
					IF FIND(fbFileGet.sLine,'>') = 0 THEN sLine := fbFileGet.sLine; END_IF	
						bRestOfDescriptionInNextLine := FALSE; 
							sLineRest := '';
								iStateParseDocument := 3; fbfileGet.bExecute := FALSE; byCounterWaitInStep := 0;
			END_IF
				IF bNotGet AND iStateParseDocument = 2 THEN
					sLine := MID(fbFileGet.sLine,255 - FIND(fbFileGet.sLine,'>'),FIND(fbFileGet.sLine,'>') + 1);
						bNotGet := FALSE;
							iStateParseDocument := 3;
								byCounterWaitInStep := 0;
				END_IF
		
		IF (timTimout.Q AND NOT fbFileGet.bEOF) OR FPErrorGet.Q THEN iStateParseDocument := 200; END_IF 
			IF FPErrorGet.Q THEN udiErrorCode := 106; END_IF
				IF timTimout.Q AND NOT fbFileGet.bEOF THEN udiErrorCode := 100; END_IF 
	
	3://Check position in file
		fbFileTell.bExecute := TRUE;

		byCounterWaitInStep := byCounterWaitInStep + 1;
		
		IF NOT fbFileTell.bBusy AND NOT fbFileTell.bError AND byCounterWaitInStep >= 2 THEN iStateParseDocument := 4; fbFileTell.bExecute := FALSE; byCounterWaitInStep := 0; END_IF
					
		IF (timTimout.Q AND NOT fbFileGet.bEOF) OR FPErrorTell.Q THEN iStateParseDocument := 200; END_IF 
			IF FPErrorTell.Q THEN udiErrorCode := 113; END_IF
				IF timTimout.Q AND NOT fbFileGet.bEOF THEN udiErrorCode := 100; END_IF 			
	
	4://Check the content what is writen between <>
		iFindBegin := FIND(sLine,'<');
			iFindEnd := FIND(sLine,'>'); 
		
		bDeleteStep3 := FALSE;	
			
		//Complete content is in 1 line	
		IF ((iFindBegin <> 0 OR iFindEnd <> 0) AND iFindEnd > iFindBegin) THEN
			IF NOT bNoNewDescription THEN sDescription := MID(sLine,iFindEnd - iFindBegin - 1,iFindBegin + 1); END_IF
				//Name from big data 
				IF ((FIND(sDescription,'Name Namespace="') <> 0 OR sDescription = 'Name') AND NOT bSymbolNameFound) THEN
					//Workaround when we use Big Data from library. Because then its writen before allways Namespace
					IF FIND(sDescription,'Name Namespace="') <> 0 THEN sDescription := 'Name'; END_IF 
						iStateParseDocument := 5;
							IF NOT bNoNewDescription THEN sLine := DELETE(sLine,iFindEnd,1); END_IF
								bNoNewDescription := FALSE;
				//Subitem (struct and FB)
				ELSIF (FIND(sDescription,'Name Namespace="') <> 0 OR sDescription = 'Name' OR sDescription = 'Type' OR FIND(sDescription,'Type Namespace="') <> 0 OR sDescription = 'Comment' OR sDescription = 'Value' OR sDescription = 'LBound' OR sDescription = 'Elements') AND bSymbolNameFound AND NOT bEnumDetected THEN 
					//Workaround when we use Structure or FB from library. Because then its writen before allways Namespace
					IF FIND(sDescription,'Name Namespace="') <> 0 THEN sDescription := 'Name'; END_IF 
					IF FIND(sDescription,'Type Namespace="') <> 0 THEN sDescription := 'Type'; END_IF
						iStateParseDocument := 6;
							IF NOT bNoNewDescription THEN sLine := DELETE(sLine,iFindEnd,1); END_IF
								bNoNewDescription := FALSE;
									bFBOrStructDetected := TRUE;
				//Subitem (Enum)
				ELSIF (sDescription = 'Text' OR sDescription = 'Enum' OR sDescription = 'Comment') AND bSymbolNameFound AND NOT bFBOrStructDetected THEN 
					iStateParseDocument := 6;
						IF NOT bNoNewDescription THEN sLine := DELETE(sLine,iFindEnd,1); END_IF
							bNoNewDescription := FALSE;
								bEnumDetected := TRUE;
									sLBound := ''; sElements := ''; uiDimensionArray := 0;
				//End of the big data
				ELSIF sDescription = '/DataType' AND bSymbolNameFound THEN 
					iStateParseDocument := 8;
				ELSE 
					sLine := DELETE(sLine,iFindEnd,1); 
						bDeleteStep3 := TRUE;
			 	END_IF
		END_IF
			//Content is not received in 1 line or nor begin no end is detected
			IF (iFindBegin <> 0 AND iFindEnd = 0) OR (iFindBegin = 0 AND iFindEnd = 0) THEN
				sLineRest := sLine;
					bRestOfDescriptionInNextLine := TRUE;
						IF NOT fbfileGet.bEOF THEN iStateParseDocument := 2; END_IF
			END_IF
				//Check ><
				IF iFindBegin <> 0 AND iFindEnd <> 0 AND iFindBegin = (iFindEnd + 1) THEN
					sLine := DELETE(sLine,FIND(sLine,'>'),1);
						bRestOfDescriptionInNextLine := FALSE; 
				END_IF
					//Check no needed description
					IF ((sDescription <> 'Name' OR sDescription <> 'Type' OR sDescription <> 'Comment' OR sDescription <> 'Text' OR sDescription <> 'Enum' OR sDescription = 'Value' OR sDescription = 'LBound' OR sDescription = 'Elements') AND iStateParseDocument = 4 AND NOT bDeleteStep3) THEN
						sLine := DELETE(sLine,FIND(sLine,'>'),1);	
					END_IF
						//Line is done
						IF LEN(sLine) = 0 AND iStateParseDocument = 4 AND NOT fbfileGet.bEOF THEN iStateParseDocument := 2; END_IF
		
		//If bEOF is True then after Timeout Line is complete
		IF timTimout.Q AND fbFileGet.bEOF THEN iStateParseDocument := 100; END_IF
			IF timTimout.Q AND NOT fbFileGet.bEOF THEN iStateParseDocument := 200; udiErrorCode := 100; END_IF	
		
	5://Check first the symbol type in document
		iFindBegin := FIND(sLine,'<');
			iFindEnd := FIND(sLine,'>'); 
		
		//Name from the symbol is not received in 1 line
		IF iFindBegin = 0 OR iFindEnd = 0 THEN
			sLineRest := sLine;
				bRestOfDescriptionInNextLine := TRUE;
					bNoNewDescription := TRUE;
						IF NOT fbfileGet.bEOF THEN iStateParseDocument := 2; END_IF
		END_IF
			//Name from the symbol is in 1 line
			IF iFindBegin <> 0 AND sDescription = 'Name' AND iStateParseDocument = 5 THEN
				sSymbolName := LEFT(sLine,iFindBegin - 1);
					sLine := DELETE(sLine,iFindBegin - 1,1);
						iStateParseDocument := 4;
							bSymbolNameFound := TRUE;
								bRestOfDescriptionInNextLine := FALSE;
			END_IF 
				//Line is done
				IF LEN(sLine) = 0 AND iStateParseDocument = 5 AND NOT fbfileGet.bEOF THEN iStateParseDocument := 2; END_IF	
		
		//If bEOF is True then after Timeout Line is complete
		IF timTimout.Q AND fbFileGet.bEOF THEN iStateParseDocument := 100; END_IF
			IF timTimout.Q AND NOT fbFileGet.bEOF THEN iStateParseDocument := 200; udiErrorCode := 100; END_IF
						
	6://Check the Sub Items
		iFindBegin := FIND(sLine,'<');
			iFindEnd := FIND(sLine,'>'); 
				iFindBeginComment := FIND(sLine,'[');
					iFindEndComment := FIND(sLine,']]');
					
		//Check they are more than Constants_Communicator.uiArraySizeOfMarkedSubItems symbols in the subitems			
		IF uiSubItemArrayInProgress > Constants_Communicator.uiArraySizeOfMarkedSubItems THEN iStateParseDocument := 200; udiErrorCode := 103; END_IF 			
			uiSubItemArrayInProgress := LIMIT(1,uiSubItemArrayInProgress,Constants_Communicator.uiArraySizeOfMarkedSubItems); 
		
		//Content from Sub Item is not received in 1 line
		IF iFindBegin = 0 OR iFindEnd = 0 AND iStateParseDocument = 6 THEN
			sLineRest := sLine;
				bRestOfDescriptionInNextLine := TRUE;
					bNoNewDescription := TRUE;
						IF NOT fbfileGet.bEOF THEN iStateParseDocument := 2; END_IF
		END_IF
			//Content from SubItem is in 1 line (FB or struct)
			IF iFindBegin <> 0 AND bFBOrStructDetected AND iStateParseDocument = 6 AND (sDescription = 'Name' OR sDescription = 'Type' OR sDescription = 'Comment' OR sDescription = 'Value' OR sDescription = 'LBound' OR sDescription = 'Elements') THEN
				IF sDescription = 'Name' AND sSymbolName <> '' THEN sNameSubItem := LEFT(sLine,(iFindBegin - 1)); END_IF
				IF sDescription = 'Type' AND sSymbolName <> '' THEN sTypeSubItem := LEFT(sLine,(iFindBegin - 1)); END_IF	
				IF sDescription = 'Comment' AND sSymbolName <> '' THEN
					sComment := MID(sLine,iFindEndComment - iFindBeginComment,iFindBeginComment + 7);
						iFindEndComment := FIND(sComment,']]');
							iLenghComment := LEN(sComment);
								sUnit := MID(sComment,(FIND(sComment,')') - FIND(sComment,'(')) - 1,FIND(sComment,'(') + 1);	
									sComment := DELETE(sComment,iLenghComment - iFindEndComment + 1,iFindEndComment);	
				END_IF
				IF sDescription = 'Value' AND sSymbolName <> '' THEN sValue := MID(sLine,iFindBegin - 1,FIND(sLine,'F')); END_IF
				IF sDescription = 'LBound' AND sSymbolName <> '' THEN sLBound := LEFT(sLine,(iFindBegin - 1)); END_IF
				IF sDescription = 'Elements' AND sSymbolName <> '' THEN sElements := LEFT(sLine,(iFindBegin - 1)); END_IF 
					sLine := DELETE(sLine,iFindBegin - 1,1);
						IF iStateParseDocument = 6 THEN iStateParseDocument := 7; END_IF
							bRestOfDescriptionInNextLine := FALSE;
			END_IF 
				//Content from SubItem is in 1 line (Enum)
				IF iFindBegin <> 0 AND bEnumDetected AND iStateParseDocument = 6 AND (sDescription = 'Text' OR sDescription = 'Enum' OR sDescription = 'Comment') THEN
					IF sDescription = 'Text' AND sSymbolName <> '' THEN sTextEnum := LEFT(sLine,(iFindBegin - 1)); END_IF
					IF sDescription = 'Enum' AND sSymbolName <> '' THEN sIndexEnum := LEFT(sLine,(iFindBegin - 1)); END_IF
					IF sDescription = 'Comment' AND sSymbolName <> '' THEN
						sComment := MID(sLine,iFindEndComment - iFindBeginComment,iFindBeginComment + 7);
							iFindEndComment := FIND(sComment,']]');
								iLenghComment := LEN(sComment);
									sUnit := MID(sComment,(FIND(sComment,')') - FIND(sComment,'(')) - 1,FIND(sComment,'(') + 1);
										sComment := DELETE(sComment,iLenghComment - iFindEndComment + 1,iFindEndComment);	 
					END_IF 
						sLine := DELETE(sLine,iFindBegin - 1,1);
							IF iStateParseDocument = 6 THEN iStateParseDocument := 7; END_IF
								bRestOfDescriptionInNextLine := FALSE;
				END_IF
					//Line is done
					IF LEN(sLine) = 0 AND iStateParseDocument = 6 AND NOT fbfileGet.bEOF THEN iStateParseDocument := 2; END_IF

		//If bEOF is True then after Timeout Line is complete
		IF timTimout.Q AND fbFileGet.bEOF THEN iStateParseDocument := 100; END_IF
			IF timTimout.Q AND NOT fbFileGet.bEOF THEN iStateParseDocument := 200; udiErrorCode := 100; END_IF		
	
	7://Check the comment
		//Clear Array information if a new SubItem Name is in progress
		IF sNameSubItem <> sNameSubItemOld THEN sLBound := ''; sElements := ''; uiDimensionArray := 0; sNameSubItemOld := sNameSubItem; END_IF 
	
		//Ckeck for multi-dimensional arrays
		IF sLBound <> '' AND sElements <> '' THEN uiDimensionArray := uiDimensionArray + 1; END_IF
		
		//Struct detected
		IF (((sSymbolName <> '' AND sNameSubItem <> '' AND sTypeSubItem <> '' AND sComment <> '' AND sSymbolName <> TwinCAT_SystemInfoVarList._AppInfo.ProjectName) OR (sSymbolName <> '' AND sNameSubItem <> '' AND sTypeSubItem <> '' AND sLBound <> '' AND sElements <> '' AND sComment <> '' AND sSymbolName <> TwinCAT_SystemInfoVarList._AppInfo.ProjectName)) AND bFBOrStructDetected) THEN
			IF MID(sComment,14,1) = '{#lynus.ag#()}' THEN 
				IF LEN(sSymbolName) <= 48 AND LEN(sNameSubItem) <= 48 THEN
					arrContentOfDocument[uiCounterWantedSymbolInProgress].sSymbolName := sSymbolName;
			 			arrContentOfDocument[uiCounterWantedSymbolInProgress].arrSubItemName[uiSubItemArrayInProgress] := sNameSubItem;
							arrContentOfDocument[uiCounterWantedSymbolInProgress].arrSubItemSymbolType[uiSubItemArrayInProgress] := sTypeSubItem;
								arrContentOfDocument[uiCounterWantedSymbolInProgress].eSymbolType := eSymbolTypeFromDocument.eIsStruct;
									arrContentOfDocument[uiCounterWantedSymbolInProgress].arrSubItemUnit[uiSubItemArrayInProgress] := sUnit;	
									//Ckeck the lenght from the String
									IF FIND(arrContentOfDocument[uiCounterWantedSymbolInProgress].arrSubItemSymbolType[uiSubItemArrayInProgress],'STRING(') <> 0 OR FIND(arrContentOfDocument[uiCounterWantedSymbolInProgress].arrSubItemSymbolType[uiSubItemArrayInProgress],'OF STRING(') <> 0 THEN
										uliSizeOfString := STRING_TO_ULINT(MID(arrContentOfDocument[uiCounterWantedSymbolInProgress].arrSubItemSymbolType[uiSubItemArrayInProgress],FIND(arrContentOfDocument[uiCounterWantedSymbolInProgress].arrSubItemSymbolType[uiSubItemArrayInProgress],')') - 
															FIND(arrContentOfDocument[uiCounterWantedSymbolInProgress].arrSubItemSymbolType[uiSubItemArrayInProgress],'(') - 1,FIND(arrContentOfDocument[uiCounterWantedSymbolInProgress].arrSubItemSymbolType[uiSubItemArrayInProgress],'(') + 1));
										IF uliSizeOfString <> 30 THEN iStateParseDocument := 200; udiErrorCode := 112; END_IF
									END_IF  
										//Check the size from the array
										IF sElements <> '' AND sLBound <> '' AND (TO_ULINT(sElements) - TO_ULINT(sLBound)) + 1 <= Constants_Communicator.bySizeOfValueArray THEN 
											arrContentOfDocument[uiCounterWantedSymbolInProgress].arrSubItemSymbolType[uiSubItemArrayInProgress] := 
												CONCAT(CONCAT('ARRAY [',sLBound),CONCAT(CONCAT('..',sElements),CONCAT('] OF ',arrContentOfDocument[uiCounterWantedSymbolInProgress].arrSubItemSymbolType[uiSubItemArrayInProgress])));
										END_IF
											IF (sElements <> '' AND sLBound <> '' AND (TO_ULINT(sElements) - TO_ULINT(sLBound)) + 1 > Constants_Communicator.bySizeOfValueArray) OR uiDimensionArray > 2 THEN
												iStateParseDocument := 200; 
													udiErrorCode := 111;
											END_IF
												//Commetn to long
												IF LEN(sUnit) > 240 OR LEN2(ADR(sComment)) > 255 THEN udiErrorCode := 3; iStateParseDocument := 200; END_IF  
												//Comment is worng
												IF LEN(sComment) > 14 AND MID(sComment,3,15) <> ' //' THEN udiErrorCode := 4; iStateParseDocument := 200; END_IF  			  
					uiSubItemArrayInProgress := uiSubItemArrayInProgress + 1;
						IF iStateParseDocument = 7 THEN 
							iStateParseDocument := 4; 
								sNameSubItem := '';
									sTypeSubItem := '';
										sComment := '';
											sLBound := '';
												sElements := '';
													uliSizeOfString := 0;
														bWaitForFB := TRUE;
															sUnit := '';
						END_IF
				ELSE
					IF LEN(sSymbolName) > 48 THEN iStateParseDocument := 200; udiErrorCode := 102; END_IF
					IF LEN(sNameSubItem) > 48 THEN iStateParseDocument := 200; udiErrorCode := 104; END_IF
				END_IF
			END_IF
		END_IF
			//FB detected
			IF sSymbolName <> '' AND sSymbolName <> TwinCAT_SystemInfoVarList._AppInfo.ProjectName AND sValue = 'FunctionBlock' AND bWaitForFB AND bFBOrStructDetected THEN
				arrContentOfDocument[uiCounterWantedSymbolInProgress].eSymbolType := eSymbolTypeFromDocument.eIsFunctionBlock; 	
					IF iStateParseDocument = 7 THEN 
						iStateParseDocument := 4; 
							sValue := '';
					END_IF
			END_IF
				//Enum detected
				IF sSymbolName <> '' AND sTextEnum <> '' AND sIndexEnum <> '' AND sComment <> '' AND sSymbolName <> TwinCAT_SystemInfoVarList._AppInfo.ProjectName AND bEnumDetected THEN
					IF MID(sComment,14,1) = '{#lynus.ag#()}' THEN 
						IF LEN(sSymbolName) <= 48 AND LEN(sTextEnum) <= 48 AND LEN(sIndexEnum) <= 6 THEN
							arrContentOfDocument[uiCounterWantedSymbolInProgress].sSymbolName := sSymbolName;
								arrContentOfDocument[uiCounterWantedSymbolInProgress].arrSubItemTextEnum[uiSubItemArrayInProgress] := sTextEnum;
									arrContentOfDocument[uiCounterWantedSymbolInProgress].arrSubItemIndexEnum[uiSubItemArrayInProgress] := sIndexEnum;
										arrContentOfDocument[uiCounterWantedSymbolInProgress].eSymbolType := eSymbolTypeFromDocument.eIsEnum;	
											arrContentOfDocument[uiCounterWantedSymbolInProgress].arrSubItemUnit[uiSubItemArrayInProgress] := sUnit;	
												//Commetn to long
												IF LEN(sUnit) > 240 OR LEN2(ADR(sComment)) > 255 THEN udiErrorCode := 3; iStateParseDocument := 200; END_IF 
												//Comment is worng
												IF LEN(sComment) > 14 AND MID(sComment,3,15) <> ' //' THEN udiErrorCode := 4; iStateParseDocument := 200; END_IF	
							uiSubItemArrayInProgress := uiSubItemArrayInProgress + 1;
								IF iStateParseDocument = 7 THEN 
									iStateParseDocument := 4;
										sComment := '';
											sTextEnum := '';
												sIndexEnum := '';
													sUnit := '';
								END_IF
						ELSE
							IF LEN(sSymbolName) > 48 THEN iStateParseDocument := 200; udiErrorCode := 102; END_IF
							IF LEN(sTextEnum) > 48 THEN iStateParseDocument := 200; udiErrorCode := 109; END_IF
							IF LEN(sIndexEnum) > 6 THEN iStateParseDocument := 200; udiErrorCode := 110; END_IF
						END_IF
					END_IF
				END_IF
				
		IF iStateParseDocument = 7 THEN iStateParseDocument := 4; END_IF
		
		//If bEOF is True then after Timeout Line is complete
		IF timTimout.Q AND fbFileGet.bEOF THEN iStateParseDocument := 100; END_IF
			IF timTimout.Q AND NOT fbFileGet.bEOF THEN iStateParseDocument := 200; udiErrorCode := 100; END_IF
		
	8://End of Datatype
		IF sDescription = '/DataType' THEN
			sLine := DELETE(sLine,FIND(sLine,'>'),1);
				IF arrContentOfDocument[uiCounterWantedSymbolInProgress].sSymbolName <> '' THEN uiCounterWantedSymbolInProgress := uiCounterWantedSymbolInProgress + 1; END_IF
					IF uiCounterWantedSymbolInProgress > Constants_Communicator.uiArraySizeOfSubItems  THEN iStateParseDocument := 200; udiErrorCode := 108; END_IF
						sSymbolName := '';
							sValue := '';
								sLBound := '';
									sElements := '';
										uiSubItemArrayInProgress := 0;
											bSymbolNameFound := FALSE;
												bFBOrStructDetected := FALSE;
													bEnumDetected := FALSE;
														bWaitForFB := FALSE; 
															uiDimensionArray := 0;
																IF iStateParseDocument = 8 THEN iStateParseDocument := 4; END_IF
		END_IF		
			
		//If bEOF is True then after Timeout Line is complete
		IF timTimout.Q AND fbFileGet.bEOF THEN iStateParseDocument := 100; END_IF
			IF timTimout.Q AND NOT fbFileGet.bEOF THEN iStateParseDocument := 200; udiErrorCode := 100; END_IF
		
	100://Close file
		fbFileClose.bExecute := TRUE;

		byCounterWaitInStep := byCounterWaitInStep + 1; 
		
		IF NOT fbFileClose.bBusy AND NOT fbFileClose.bError AND byCounterWaitInStep >= 2 THEN iStateParseDocument := 101; fbFileClose.bExecute := FALSE; byCounterWaitInStep := 0; END_IF	
		
		IF (timTimout.Q AND NOT fbFileGet.bEOF) OR FPErrorClose.Q THEN iStateParseDocument := 200; END_IF
			IF FPErrorClose.Q THEN udiErrorCode := 107; END_IF 
				IF timTimout.Q AND NOT fbFileGet.bEOF THEN udiErrorCode := 100; END_IF 
		
	101://Search all "No Standart" Data Types that occur in the FB and structures Step 1 (Its solved with counter and not with a loop because the code must work also on a small plc) (Start with progress + 1)
		uiCounterFBorStruct := uiCounterFBorStruct + 1; 
			IF uiCounterFBorStruct > Constants_Communicator.uiArraySizeOfMarkedSubItems THEN uiCounterInProgressFromDocument := uiCounterInProgressFromDocument + 1; uiCounterFBorStruct := 1; END_IF
				uiCounterInProgressFromDocument := LIMIT(1,uiCounterInProgressFromDocument,Constants_Communicator.uiArraySizeOfSubItems);
		
		IF ((arrContentOfDocument[uiCounterInProgressFromDocument].eSymbolType = eSymbolTypeFromDocument.eIsFunctionBlock OR arrContentOfDocument[uiCounterInProgressFromDocument].eSymbolType = eSymbolTypeFromDocument. eIsStruct) AND arrContentOfDocument[1].sSymbolName <> '') THEN
			IF arrContentOfDocument[uiCounterInProgressFromDocument].arrSubItemSymbolType[uiCounterFBorStruct] <> 'BOOL' AND arrContentOfDocument[uiCounterInProgressFromDocument].arrSubItemSymbolType[uiCounterFBorStruct] <> 'BYTE' AND
				arrContentOfDocument[uiCounterInProgressFromDocument].arrSubItemSymbolType[uiCounterFBorStruct] <> 'WORD' AND arrContentOfDocument[uiCounterInProgressFromDocument].arrSubItemSymbolType[uiCounterFBorStruct] <> 'DWORD' AND
					arrContentOfDocument[uiCounterInProgressFromDocument].arrSubItemSymbolType[uiCounterFBorStruct] <> 'SINT' AND arrContentOfDocument[uiCounterInProgressFromDocument].arrSubItemSymbolType[uiCounterFBorStruct] <> 'USINT' AND
						arrContentOfDocument[uiCounterInProgressFromDocument].arrSubItemSymbolType[uiCounterFBorStruct] <> 'INT' AND arrContentOfDocument[uiCounterInProgressFromDocument].arrSubItemSymbolType[uiCounterFBorStruct] <> 'UINT' AND
							arrContentOfDocument[uiCounterInProgressFromDocument].arrSubItemSymbolType[uiCounterFBorStruct] <> 'DINT' AND arrContentOfDocument[uiCounterInProgressFromDocument].arrSubItemSymbolType[uiCounterFBorStruct] <> 'UDINT' AND
								arrContentOfDocument[uiCounterInProgressFromDocument].arrSubItemSymbolType[uiCounterFBorStruct] <> 'LINT' AND arrContentOfDocument[uiCounterInProgressFromDocument].arrSubItemSymbolType[uiCounterFBorStruct] <> 'ULINT' AND
									arrContentOfDocument[uiCounterInProgressFromDocument].arrSubItemSymbolType[uiCounterFBorStruct] <> 'LWORD' AND arrContentOfDocument[uiCounterInProgressFromDocument].arrSubItemSymbolType[uiCounterFBorStruct] <> 'REAL' AND
										arrContentOfDocument[uiCounterInProgressFromDocument].arrSubItemSymbolType[uiCounterFBorStruct] <> 'LREAL' AND arrContentOfDocument[uiCounterInProgressFromDocument].arrSubItemSymbolType[uiCounterFBorStruct] <> 'STRING(30)' AND
											arrContentOfDocument[uiCounterInProgressFromDocument].arrSubItemSymbolType[uiCounterFBorStruct] <> 'TIME' AND arrContentOfDocument[uiCounterInProgressFromDocument].arrSubItemSymbolType[uiCounterFBorStruct] <> 'TIME_OF_DAY' AND
												arrContentOfDocument[uiCounterInProgressFromDocument].arrSubItemSymbolType[uiCounterFBorStruct] <> 'DATE' AND arrContentOfDocument[uiCounterInProgressFromDocument].arrSubItemSymbolType[uiCounterFBorStruct] <> 'DATE_AND_TIME' AND  
			FIND(arrContentOfDocument[uiCounterInProgressFromDocument].arrSubItemSymbolType[uiCounterFBorStruct],'OF BOOL') = 0 AND FIND(arrContentOfDocument[uiCounterInProgressFromDocument].arrSubItemSymbolType[uiCounterFBorStruct],'OF BYTE') = 0 AND
				FIND(arrContentOfDocument[uiCounterInProgressFromDocument].arrSubItemSymbolType[uiCounterFBorStruct],'OF WORD') = 0 AND FIND(arrContentOfDocument[uiCounterInProgressFromDocument].arrSubItemSymbolType[uiCounterFBorStruct],'OF DWORD') = 0 AND
					FIND(arrContentOfDocument[uiCounterInProgressFromDocument].arrSubItemSymbolType[uiCounterFBorStruct],'OF SINT') = 0 AND FIND(arrContentOfDocument[uiCounterInProgressFromDocument].arrSubItemSymbolType[uiCounterFBorStruct],'OF USINT') = 0 AND 
						FIND(arrContentOfDocument[uiCounterInProgressFromDocument].arrSubItemSymbolType[uiCounterFBorStruct],'OF INT') = 0 AND FIND(arrContentOfDocument[uiCounterInProgressFromDocument].arrSubItemSymbolType[uiCounterFBorStruct],'OF UINT') = 0 AND
							FIND(arrContentOfDocument[uiCounterInProgressFromDocument].arrSubItemSymbolType[uiCounterFBorStruct],'OF DINT') = 0 AND FIND(arrContentOfDocument[uiCounterInProgressFromDocument].arrSubItemSymbolType[uiCounterFBorStruct],'OF UDINT') = 0 AND
								FIND(arrContentOfDocument[uiCounterInProgressFromDocument].arrSubItemSymbolType[uiCounterFBorStruct],'OF LINT') = 0 AND FIND(arrContentOfDocument[uiCounterInProgressFromDocument].arrSubItemSymbolType[uiCounterFBorStruct],'OF ULINT') = 0 AND
									FIND(arrContentOfDocument[uiCounterInProgressFromDocument].arrSubItemSymbolType[uiCounterFBorStruct],'OF LWORD') = 0 AND FIND(arrContentOfDocument[uiCounterInProgressFromDocument].arrSubItemSymbolType[uiCounterFBorStruct],'OF REAL') = 0 AND
										FIND(arrContentOfDocument[uiCounterInProgressFromDocument].arrSubItemSymbolType[uiCounterFBorStruct],'OF LREAL') = 0 AND FIND(arrContentOfDocument[uiCounterInProgressFromDocument].arrSubItemSymbolType[uiCounterFBorStruct],'OF STRING(30)') = 0 AND
											FIND(arrContentOfDocument[uiCounterInProgressFromDocument].arrSubItemSymbolType[uiCounterFBorStruct],'OF TIME') = 0 AND FIND(arrContentOfDocument[uiCounterInProgressFromDocument].arrSubItemSymbolType[uiCounterFBorStruct],'OF TIME_OF_DAY') = 0 AND
												FIND(arrContentOfDocument[uiCounterInProgressFromDocument].arrSubItemSymbolType[uiCounterFBorStruct],'OF DATE') = 0 AND FIND(arrContentOfDocument[uiCounterInProgressFromDocument].arrSubItemSymbolType[uiCounterFBorStruct],'OF DATE_AND_TIME') = 0 AND
													FIND(arrContentOfDocument[uiCounterInProgressFromDocument].arrSubItemSymbolType[uiCounterFBorStruct],'ARRAY') = 0 AND
				arrContentOfDocument[uiCounterInProgressFromDocument].arrSubItemSymbolType[uiCounterFBorStruct] <> '' THEN
					uiCounterListForFBorStruct := uiCounterListForFBorStruct + 1;
						uiCounterListForFBorStruct := LIMIT(1,uiCounterListForFBorStruct,Constants_Communicator.uiArraySizeOfSubItems);
							arrNumberForLPCheckIdentSymbols[1] := Constants_Communicator.uiArraySizeOfSubItems / 4;
							arrNumberForLPCheckIdentSymbols[2] := Constants_Communicator.uiArraySizeOfSubItems / 4;
							arrNumberForLPCheckIdentSymbols[3] := Constants_Communicator.uiArraySizeOfSubItems / 4;
							arrNumberForLPCheckIdentSymbols[4] := Constants_Communicator.uiArraySizeOfSubItems - arrNumberForLPCheckIdentSymbols[1] - arrNumberForLPCheckIdentSymbols[2] - arrNumberForLPCheckIdentSymbols[3]; 
								iStateParseDocument := 102;	
			END_IF		
		END_IF
	
		IF (((uiCounterInProgressFromDocument >= (uiCounterWantedSymbolInProgress - 1)) AND iStateParseDocument = 101 AND uiCounterFBorStruct >= Constants_Communicator.uiArraySizeOfMarkedSubItems AND 
			(arrContentOfDocument[uiCounterInProgressFromDocument].eSymbolType = eSymbolTypeFromDocument.eIsFunctionBlock OR arrContentOfDocument[uiCounterInProgressFromDocument].eSymbolType = eSymbolTypeFromDocument. eIsStruct))) OR 
				((uiCounterInProgressFromDocument >= (uiCounterWantedSymbolInProgress - 1)) AND iStateParseDocument = 101 AND 
					arrContentOfDocument[uiCounterInProgressFromDocument].eSymbolType <> eSymbolTypeFromDocument.eIsFunctionBlock AND arrContentOfDocument[uiCounterInProgressFromDocument].eSymbolType <> eSymbolTypeFromDocument. eIsStruct) OR
						arrContentOfDocument[1].sSymbolName = '' OR uiCounterWantedSymbolInProgress = 1 THEN
							iStateParseDocument := 103;
								byProgress := byProgress + 1;
		END_IF
			IF arrContentOfDocument[uiCounterInProgressFromDocument].eSymbolType <> eSymbolTypeFromDocument.eIsFunctionBlock AND arrContentOfDocument[uiCounterInProgressFromDocument].eSymbolType <> eSymbolTypeFromDocument. eIsStruct AND 
				iStateParseDocument = 101 THEN
					uiCounterInProgressFromDocument := uiCounterInProgressFromDocument + 1;
			END_IF	
		
	102://Search all "No Standart" Data Types that occur in the FB and structures Step 2
		byCounterWaitInStep := byCounterWaitInStep + 1;
	
		IF byCounterWaitInStep = 1 THEN
			FOR uiLPCheckIdentSymbols := 1 TO arrNumberForLPCheckIdentSymbols[1] BY 1 DO 
				IF arrCheckListForNestedSymbols[uiLPCheckIdentSymbols] = arrContentOfDocument[uiCounterInProgressFromDocument].arrSubItemSymbolType[uiCounterFBorStruct] THEN 
					uiCounterListForFBorStruct := uiCounterListForFBorStruct - 1;
						byCounterWaitInStep := 5;
							EXIT;
				END_IF
			END_FOR
		END_IF
			IF byCounterWaitInStep = 2 THEN
				FOR uiLPCheckIdentSymbols := arrNumberForLPCheckIdentSymbols[1] TO arrNumberForLPCheckIdentSymbols[1] + arrNumberForLPCheckIdentSymbols[2] BY 1 DO 
					IF arrCheckListForNestedSymbols[uiLPCheckIdentSymbols] = arrContentOfDocument[uiCounterInProgressFromDocument].arrSubItemSymbolType[uiCounterFBorStruct] THEN 
						uiCounterListForFBorStruct := uiCounterListForFBorStruct - 1;
							byCounterWaitInStep := 5;
								EXIT;
					END_IF
				END_FOR
			END_IF
				IF byCounterWaitInStep = 3 THEN
					FOR uiLPCheckIdentSymbols := arrNumberForLPCheckIdentSymbols[1] + arrNumberForLPCheckIdentSymbols[2] TO arrNumberForLPCheckIdentSymbols[1] + arrNumberForLPCheckIdentSymbols[2] + arrNumberForLPCheckIdentSymbols[3] BY 1 DO 
						IF arrCheckListForNestedSymbols[uiLPCheckIdentSymbols] = arrContentOfDocument[uiCounterInProgressFromDocument].arrSubItemSymbolType[uiCounterFBorStruct] THEN 
							uiCounterListForFBorStruct := uiCounterListForFBorStruct - 1;
								byCounterWaitInStep := 5;
									EXIT;
						END_IF
					END_FOR
				END_IF
					IF byCounterWaitInStep = 4 THEN
						FOR uiLPCheckIdentSymbols := arrNumberForLPCheckIdentSymbols[1] + arrNumberForLPCheckIdentSymbols[2] + arrNumberForLPCheckIdentSymbols[3] TO arrNumberForLPCheckIdentSymbols[1] + arrNumberForLPCheckIdentSymbols[2] + arrNumberForLPCheckIdentSymbols[3] + arrNumberForLPCheckIdentSymbols[4] BY 1 DO 
							IF arrCheckListForNestedSymbols[uiLPCheckIdentSymbols] = arrContentOfDocument[uiCounterInProgressFromDocument].arrSubItemSymbolType[uiCounterFBorStruct] THEN 
								uiCounterListForFBorStruct := uiCounterListForFBorStruct - 1;
									EXIT;
							ELSIF uiLPCheckIdentSymbols >= arrNumberForLPCheckIdentSymbols[1] + arrNumberForLPCheckIdentSymbols[2] + arrNumberForLPCheckIdentSymbols[3] + arrNumberForLPCheckIdentSymbols[4] THEN    
								arrCheckListForNestedSymbols[uiCounterListForFBorStruct] := arrContentOfDocument[uiCounterInProgressFromDocument].arrSubItemSymbolType[uiCounterFBorStruct]; 
							END_IF
						END_FOR
					END_IF	
	
		IF byCounterWaitInStep >= 4 AND (uiCounterInProgressFromDocument < (uiCounterWantedSymbolInProgress - 1)) OR 
			(byCounterWaitInStep >= 4 AND (uiCounterInProgressFromDocument = (uiCounterWantedSymbolInProgress - 1)) AND uiCounterFBorStruct < Constants_Communicator.uiArraySizeOfMarkedSubItems) THEN 
				iStateParseDocument := 101;
					byCounterWaitInStep := 0; 
		END_IF
			IF ((uiCounterInProgressFromDocument >= (uiCounterWantedSymbolInProgress - 1)) AND iStateParseDocument = 102 AND byCounterWaitInStep >= 4 AND uiCounterFBorStruct >= Constants_Communicator.uiArraySizeOfMarkedSubItems) THEN
				iStateParseDocument := 103;
					byProgress := byProgress + 1;
						byCounterWaitInStep := 0;
			END_IF
	
	103://Check if all structs and enums are found that are needed for the function blocks or structs
		uiCounterCheckSubItemsInContentOfDoc := uiCounterCheckSubItemsInContentOfDoc + 1;
			uiCounterCheckSubItemsInContentOfDoc := LIMIT(1,uiCounterCheckSubItemsInContentOfDoc,Constants_Communicator.uiArraySizeOfSubItems);
		
		IF uiCounterListForFBorStruct > 0 THEN 	
			FOR uiLPCheckIdentSymbols := 1 TO Constants_Communicator.uiArraySizeOfSubItems BY 1 DO 
				IF arrCheckListForNestedSymbols[uiCounterCheckSubItemsInContentOfDoc] = arrContentOfDocument[uiLPCheckIdentSymbols].sSymbolName THEN
					EXIT;
				ELSE
					IF uiLPCheckIdentSymbols >= Constants_Communicator.uiArraySizeOfSubItems THEN 
						iStateParseDocument := 200;
							udiErrorCode := 115;
					END_IF
				END_IF 
			END_FOR
		END_IF	 
		
		IF uiCounterCheckSubItemsInContentOfDoc >= uiCounterListForFBorStruct AND uiCounterListForFBorStruct > 0 AND iStateParseDocument = 103 THEN 
			iStateParseDocument := 104; byProgress := byProgress + 1; uiCounterCheckSubItemsInContentOfDoc := 0; 
		END_IF
			IF uiCounterListForFBorStruct = 0 AND iStateParseDocument = 103 THEN iStateParseDocument := 106; byProgress := byProgress + 1; uiCounterCheckSubItemsInContentOfDoc := 0; END_IF 
			
	104://Ckeck for other Functionblocks in used Structs or Function Blocks (Its not alowed at this Version)
		uiCounterCheckSubItemsInContentOfDoc := uiCounterCheckSubItemsInContentOfDoc + 1;
			uiCounterCheckSubItemsInContentOfDoc := LIMIT(1,uiCounterCheckSubItemsInContentOfDoc,Constants_Communicator.uiArraySizeOfSubItems);
			
		IF uiCounterInProgressFromDocument <= Constants_Communicator.uiArraySizeOfSubItems THEN	
			FOR uiLPCkeckContentInSubItems := 1 TO uiCounterInProgressFromDocument BY 1 DO
				IF arrCheckListForNestedSymbols[uiCounterCheckSubItemsInContentOfDoc] = arrContentOfDocument[uiLPCkeckContentInSubItems].sSymbolName AND 
					arrContentOfDocument[uiLPCkeckContentInSubItems].eSymbolType = eSymbolTypeFromDocument.eIsFunctionBlock THEN
						iStateParseDocument := 200;
							udiErrorCode := 116;
								EXIT;	
				END_IF
			END_FOR
		END_IF
  
		IF uiCounterCheckSubItemsInContentOfDoc >= uiCounterListForFBorStruct AND iStateParseDocument = 104 THEN iStateParseDocument := 105; byProgress := byProgress + 1; uiCounterCheckSubItemsInContentOfDoc := 0; END_IF		
		
	105://Ckeck if in the subitems in the structs or Functionblocks is not more than 1 extra Subitem
		uiCounterCkeckContenInSubItems_2 := uiCounterCkeckContenInSubItems_2 + 1;
		
		IF uiCounterCkeckContenInSubItems_2 > Constants_Communicator.uiArraySizeOfMarkedSubItems THEN uiCounterCkeckContenInSubItems_1 := uiCounterCkeckContenInSubItems_1 + 1; END_IF
			
		IF uiCounterCkeckContenInSubItems_2 > Constants_Communicator.uiArraySizeOfMarkedSubItems AND uiCounterCkeckContenInSubItems_1 > uiCounterInProgressFromDocument THEN uiCounterCheckSubItemsInContentOfDoc := uiCounterCheckSubItemsInContentOfDoc + 1; END_IF	

		IF uiCounterCkeckContenInSubItems_1 > uiCounterInProgressFromDocument THEN uiCounterCkeckContenInSubItems_1 := 1; END_IF	
		IF uiCounterCkeckContenInSubItems_2 > Constants_Communicator.uiArraySizeOfMarkedSubItems THEN uiCounterCkeckContenInSubItems_2 := 1; END_IF
	
		uiCounterCkeckContenInSubItems_2 := LIMIT(1,uiCounterCkeckContenInSubItems_2,Constants_Communicator.uiArraySizeOfMarkedSubItems);	
		uiCounterCheckSubItemsInContentOfDoc := LIMIT(1,uiCounterCheckSubItemsInContentOfDoc,Constants_Communicator.uiArraySizeOfSubItems);
		uiCounterCkeckContenInSubItems_1 := LIMIT(1,uiCounterCkeckContenInSubItems_1,Constants_Communicator.uiArraySizeOfSubItems);
			
